Yaskawa INFORM job: A_ROOF_UPPER_0614_2_PAINT_14.JBI

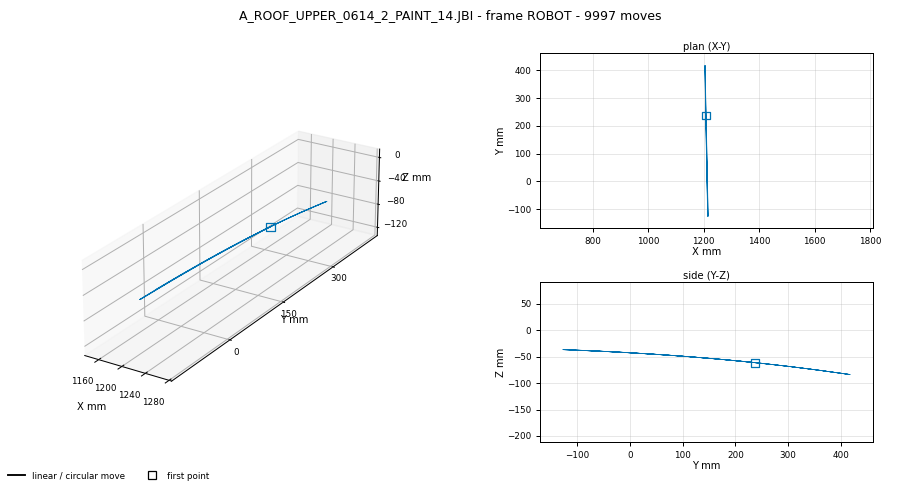
[picture p0: tool path of A_ROOF_UPPER_0614_2_PAINT_14.JBI in frame ROBOT, 9997 of 9997 moves have a stored position in this frame; points joined in program order, loops and branches not executed]
/JOB
//NAME A_ROOF_UPPER_0614_2_PAINT14
//POS
///NPOS 9997,0,0,0,0,0
///TOOL 1
///USER 0
///POSTYPE ROBOT
///RECTAN
///RCONF 1,0,0,0,0,0,0,0,0,0,0,0,0,0,0,0,0,0,0,0,0,0,0,0
C00000=1208.790,237.146,-61.145,-177.184,6.593,148.379
C00001=1208.795,236.875,-61.116,-177.187,6.591,148.380
C00002=1208.800,236.604,-61.089,-177.189,6.589,148.380
C00003=1208.804,236.355,-61.063,-177.193,6.586,148.380
C00004=1208.809,236.106,-61.037,-177.195,6.584,148.380
C00005=1208.814,235.857,-61.011,-177.197,6.582,148.381
C00006=1208.818,235.609,-60.985,-177.200,6.580,148.381
C00007=1208.823,235.360,-60.960,-177.202,6.578,148.381
C00008=1208.827,235.111,-60.934,-177.205,6.576,148.381
C00009=1208.831,234.863,-60.908,-177.207,6.575,148.382
C00010=1208.836,234.614,-60.883,-177.211,6.572,148.382
C00011=1208.840,234.366,-60.857,-177.213,6.570,148.382
C00012=1208.844,234.117,-60.831,-177.215,6.568,148.382
C00013=1208.850,233.868,-60.805,-177.218,6.566,148.383
C00014=1208.854,233.620,-60.780,-177.220,6.564,148.383
C00015=1208.858,233.371,-60.754,-177.223,6.562,148.383
C00016=1208.863,233.123,-60.728,-177.225,6.560,148.384
C00017=1208.867,232.874,-60.703,-177.228,6.558,148.384
C00018=1208.872,232.625,-60.677,-177.231,6.555,148.384
C00019=1208.876,232.377,-60.652,-177.233,6.553,148.384
C00020=1208.881,232.128,-60.626,-177.236,6.552,148.385
C00021=1208.885,231.879,-60.600,-177.239,6.550,148.385
C00022=1208.890,231.631,-60.575,-177.241,6.548,148.385
C00023=1208.894,231.383,-60.549,-177.243,6.546,148.385
C00024=1208.898,231.134,-60.523,-177.246,6.544,148.386
C00025=1208.903,230.885,-60.499,-177.248,6.542,148.386
C00026=1208.908,230.636,-60.473,-177.251,6.539,148.386
C00027=1208.912,230.387,-60.447,-177.254,6.537,148.386
C00028=1208.917,230.139,-60.422,-177.257,6.535,148.387
C00029=1208.921,229.890,-60.396,-177.259,6.533,148.387
C00030=1208.925,229.641,-60.371,-177.261,6.531,148.387
C00031=1208.930,229.393,-60.345,-177.264,6.529,148.387
C00032=1208.934,229.144,-60.320,-177.267,6.528,148.388
C00033=1208.939,228.896,-60.294,-177.269,6.526,148.388
C00034=1208.944,228.647,-60.269,-177.272,6.524,148.388
C00035=1208.948,228.398,-60.244,-177.274,6.522,148.388
C00036=1208.953,228.150,-60.218,-177.277,6.519,148.389
C00037=1208.957,227.901,-60.192,-177.280,6.517,148.389
C00038=1208.962,227.652,-60.168,-177.282,6.515,148.389
C00039=1208.966,227.403,-60.142,-177.285,6.513,148.390
C00040=1208.971,227.155,-60.117,-177.287,6.511,148.390
C00041=1208.975,226.906,-60.092,-177.290,6.510,148.390
C00042=1208.979,226.657,-60.066,-177.292,6.507,148.390
C00043=1208.984,226.409,-60.041,-177.295,6.505,148.391
C00044=1208.989,226.160,-60.016,-177.297,6.504,148.391
C00045=1208.993,225.912,-59.991,-177.300,6.502,148.391
C00046=1208.998,225.663,-59.965,-177.303,6.500,148.392
C00047=1209.003,225.414,-59.940,-177.305,6.497,148.392
C00048=1209.007,225.165,-59.914,-177.308,6.495,148.392
C00049=1209.011,224.917,-59.890,-177.311,6.493,148.392
C00050=1209.016,224.668,-59.865,-177.313,6.491,148.393
C00051=1209.020,224.419,-59.840,-177.316,6.490,148.393
C00052=1209.025,224.171,-59.814,-177.318,6.487,148.393
C00053=1209.029,223.922,-59.788,-177.321,6.486,148.393
C00054=1209.034,223.673,-59.764,-177.323,6.484,148.394
C00055=1209.038,223.425,-59.739,-177.326,6.482,148.394
C00056=1209.043,223.176,-59.714,-177.329,6.480,148.394
C00057=1209.047,222.927,-59.688,-177.331,6.478,148.394
C00058=1209.052,222.678,-59.664,-177.333,6.476,148.395
C00059=1209.056,222.429,-59.639,-177.336,6.474,148.395
C00060=1209.061,222.181,-59.614,-177.339,6.472,148.395
C00061=1209.066,221.932,-59.589,-177.342,6.470,148.396
C00062=1209.070,221.684,-59.563,-177.345,6.468,148.396
C00063=1209.075,221.435,-59.539,-177.347,6.466,148.396
C00064=1209.079,221.186,-59.513,-177.349,6.464,148.397
C00065=1209.084,220.938,-59.489,-177.352,6.462,148.397
C00066=1209.088,220.689,-59.464,-177.355,6.460,148.397
C00067=1209.093,220.440,-59.439,-177.357,6.458,148.398
C00068=1209.097,220.191,-59.414,-177.360,6.456,148.398
C00069=1209.102,219.943,-59.389,-177.362,6.454,148.398
C00070=1209.106,219.694,-59.364,-177.365,6.452,148.398
C00071=1209.111,219.445,-59.339,-177.367,6.451,148.399
C00072=1209.116,219.197,-59.314,-177.370,6.449,148.399
C00073=1209.120,218.948,-59.290,-177.373,6.447,148.399
C00074=1209.125,218.699,-59.265,-177.375,6.445,148.400
C00075=1209.128,218.450,-59.240,-177.377,6.443,148.400
C00076=1209.133,218.202,-59.215,-177.380,6.441,148.400
C00077=1209.138,217.952,-59.190,-177.383,6.438,148.400
C00078=1209.142,217.704,-59.166,-177.386,6.437,148.401
C00079=1209.147,217.455,-59.141,-177.389,6.435,148.401
C00080=1209.152,217.207,-59.116,-177.391,6.433,148.401
C00081=1209.156,216.958,-59.091,-177.394,6.431,148.402
C00082=1209.160,216.709,-59.066,-177.396,6.429,148.402
C00083=1209.165,216.460,-59.042,-177.399,6.427,148.402
C00084=1209.170,216.212,-59.017,-177.401,6.425,148.402
C00085=1209.173,215.963,-58.993,-177.404,6.423,148.403
C00086=1209.179,215.714,-58.968,-177.407,6.422,148.403
C00087=1209.184,215.466,-58.943,-177.409,6.420,148.403
C00088=1209.188,215.217,-58.919,-177.412,6.418,148.404
C00089=1209.193,214.968,-58.894,-177.414,6.416,148.404
C00090=1209.197,214.719,-58.870,-177.417,6.414,148.404
C00091=1209.201,214.471,-58.844,-177.419,6.412,148.405
C00092=1209.206,214.222,-58.820,-177.422,6.410,148.405
C00093=1209.211,213.973,-58.796,-177.425,6.408,148.405
C00094=1209.215,213.724,-58.771,-177.427,6.406,148.406
C00095=1209.220,213.476,-58.746,-177.430,6.405,148.406
C00096=1209.224,213.227,-58.722,-177.432,6.403,148.406
C00097=1209.229,212.978,-58.697,-177.435,6.401,148.407
C00098=1209.233,212.729,-58.673,-177.438,6.399,148.407
C00099=1209.238,212.481,-58.649,-177.440,6.397,148.407
C00100=1209.242,212.232,-58.624,-177.443,6.395,148.407
C00101=1209.247,211.983,-58.599,-177.445,6.393,148.408
C00102=1209.252,211.734,-58.575,-177.448,6.391,148.408
C00103=1209.257,211.464,-58.549,-177.451,6.389,148.408
C00104=1209.261,211.193,-58.522,-177.454,6.387,148.409
C00105=1209.266,210.923,-58.496,-177.456,6.385,148.409
C00106=1209.271,210.653,-58.469,-177.459,6.384,148.410
C00107=1209.276,210.404,-58.445,-177.462,6.381,148.410
C00108=1209.280,210.155,-58.420,-177.464,6.380,148.410
C00109=1209.284,209.906,-58.396,-177.467,6.378,148.410
C00110=1209.290,209.658,-58.372,-177.470,6.376,148.411
C00111=1209.294,209.409,-58.348,-177.472,6.374,148.411
C00112=1209.299,209.159,-58.323,-177.475,6.372,148.411
C00113=1209.303,208.911,-58.299,-177.477,6.370,148.412
C00114=1209.308,208.662,-58.275,-177.480,6.369,148.412
C00115=1209.313,208.414,-58.250,-177.483,6.367,148.412
C00116=1209.316,208.165,-58.226,-177.485,6.365,148.413
C00117=1209.321,207.916,-58.202,-177.488,6.363,148.413
C00118=1209.326,207.667,-58.178,-177.491,6.361,148.413
C00119=1209.331,207.418,-58.154,-177.493,6.359,148.414
C00120=1209.335,207.170,-58.130,-177.495,6.357,148.414
C00121=1209.340,206.921,-58.105,-177.498,6.355,148.414
C00122=1209.344,206.672,-58.081,-177.501,6.354,148.415
C00123=1209.349,206.423,-58.057,-177.503,6.352,148.415
C00124=1209.353,206.175,-58.033,-177.506,6.350,148.415
C00125=1209.358,205.926,-58.009,-177.509,6.348,148.416
C00126=1209.362,205.677,-57.984,-177.511,6.346,148.416
C00127=1209.367,205.428,-57.961,-177.514,6.344,148.416
C00128=1209.371,205.179,-57.937,-177.517,6.343,148.417
C00129=1209.376,204.931,-57.912,-177.519,6.341,148.417
C00130=1209.381,204.682,-57.889,-177.522,6.339,148.417
C00131=1209.385,204.433,-57.865,-177.525,6.337,148.418
C00132=1209.389,204.184,-57.840,-177.527,6.335,148.418
C00133=1209.395,203.935,-57.816,-177.530,6.333,148.418
C00134=1209.399,203.686,-57.792,-177.533,6.332,148.419
C00135=1209.404,203.437,-57.769,-177.535,6.330,148.419
C00136=1209.408,203.189,-57.745,-177.538,6.328,148.419
C00137=1209.412,202.941,-57.721,-177.540,6.326,148.420
C00138=1209.418,202.691,-57.697,-177.543,6.324,148.420
C00139=1209.422,202.443,-57.673,-177.546,6.322,148.420
C00140=1209.426,202.193,-57.649,-177.548,6.320,148.420
C00141=1209.431,201.945,-57.625,-177.551,6.319,148.421
C00142=1209.435,201.696,-57.601,-177.553,6.317,148.421
C00143=1209.440,201.447,-57.577,-177.556,6.315,148.421
C00144=1209.444,201.199,-57.553,-177.558,6.314,148.422
C00145=1209.450,200.949,-57.529,-177.561,6.312,148.422
C00146=1209.454,200.701,-57.505,-177.563,6.310,148.422
C00147=1209.459,200.452,-57.482,-177.566,6.308,148.423
C00148=1209.463,200.204,-57.458,-177.569,6.307,148.423
C00149=1209.468,199.955,-57.434,-177.571,6.305,148.424
C00150=1209.472,199.705,-57.411,-177.574,6.303,148.424
C00151=1209.476,199.456,-57.387,-177.576,6.301,148.424
C00152=1209.481,199.207,-57.363,-177.579,6.299,148.425
C00153=1209.486,198.959,-57.339,-177.582,6.297,148.425
C00154=1209.490,198.710,-57.316,-177.584,6.296,148.425
C00155=1209.495,198.462,-57.292,-177.587,6.294,148.426
C00156=1209.499,198.213,-57.268,-177.590,6.292,148.426
C00157=1209.504,197.963,-57.245,-177.592,6.290,148.426
C00158=1209.508,197.715,-57.221,-177.595,6.288,148.427
C00159=1209.513,197.466,-57.198,-177.597,6.287,148.427
C00160=1209.518,197.217,-57.174,-177.600,6.285,148.427
C00161=1209.523,196.968,-57.150,-177.602,6.284,148.428
C00162=1209.528,196.719,-57.126,-177.605,6.282,148.428
C00163=1209.532,196.471,-57.104,-177.608,6.280,148.428
C00164=1209.536,196.222,-57.079,-177.610,6.278,148.429
C00165=1209.541,195.973,-57.056,-177.613,6.276,148.429
C00166=1209.545,195.724,-57.033,-177.616,6.274,148.429
C00167=1209.550,195.476,-57.009,-177.618,6.273,148.430
C00168=1209.554,195.227,-56.985,-177.621,6.271,148.430
C00169=1209.559,194.978,-56.962,-177.624,6.269,148.430
C00170=1209.564,194.729,-56.939,-177.626,6.268,148.431
C00171=1209.568,194.480,-56.914,-177.628,6.266,148.431
C00172=1209.573,194.231,-56.891,-177.631,6.264,148.432
C00173=1209.578,193.982,-56.868,-177.634,6.263,148.432
C00174=1209.582,193.733,-56.844,-177.636,6.261,148.432
C00175=1209.587,193.484,-56.821,-177.639,6.259,148.433
C00176=1209.591,193.236,-56.797,-177.642,6.257,148.433
C00177=1209.596,192.987,-56.774,-177.644,6.255,148.433
C00178=1209.601,192.738,-56.750,-177.647,6.253,148.434
C00179=1209.605,192.489,-56.728,-177.649,6.252,148.434
C00180=1209.610,192.240,-56.704,-177.652,6.251,148.435
C00181=1209.615,191.991,-56.681,-177.655,6.249,148.435
C00182=1209.620,191.742,-56.658,-177.657,6.247,148.435
C00183=1209.624,191.493,-56.634,-177.660,6.245,148.436
C00184=1209.629,191.245,-56.610,-177.663,6.244,148.436
C00185=1209.633,190.996,-56.587,-177.665,6.242,148.436
C00186=1209.637,190.747,-56.564,-177.668,6.240,148.437
C00187=1209.642,190.498,-56.541,-177.670,6.239,148.437
C00188=1209.647,190.249,-56.518,-177.673,6.237,148.437
C00189=1209.651,190.000,-56.494,-177.675,6.235,148.438
C00190=1209.656,189.751,-56.471,-177.678,6.233,148.438
C00191=1209.661,189.503,-56.448,-177.681,6.232,148.438
C00192=1209.665,189.254,-56.425,-177.683,6.230,148.439
C00193=1209.670,189.005,-56.402,-177.686,6.228,148.439
C00194=1209.675,188.756,-56.378,-177.689,6.226,148.439
C00195=1209.679,188.507,-56.355,-177.691,6.225,148.440
C00196=1209.683,188.258,-56.332,-177.693,6.223,148.440
C00197=1209.688,188.009,-56.309,-177.696,6.222,148.441
C00198=1209.693,187.760,-56.285,-177.699,6.220,148.441
C00199=1209.698,187.512,-56.262,-177.701,6.218,148.441
C00200=1209.702,187.262,-56.240,-177.704,6.216,148.442
C00201=1209.707,187.013,-56.217,-177.707,6.215,148.442
C00202=1209.712,186.764,-56.194,-177.709,6.214,148.443
C00203=1209.716,186.516,-56.171,-177.712,6.212,148.443
C00204=1209.720,186.267,-56.148,-177.715,6.210,148.443
C00205=1209.726,186.018,-56.125,-177.717,6.208,148.444
C00206=1209.730,185.770,-56.102,-177.720,6.206,148.444
C00207=1209.735,185.500,-56.077,-177.723,6.205,148.444
C00208=1209.740,185.230,-56.052,-177.725,6.203,148.445
C00209=1209.745,184.961,-56.027,-177.728,6.201,148.445
C00210=1209.750,184.691,-56.002,-177.731,6.199,148.446
C00211=1209.755,184.442,-55.979,-177.734,6.198,148.446
C00212=1209.759,184.193,-55.956,-177.736,6.196,148.446
C00213=1209.764,183.943,-55.934,-177.738,6.195,148.447
C00214=1209.768,183.695,-55.911,-177.741,6.193,148.447
C00215=1209.773,183.446,-55.888,-177.744,6.191,148.447
C00216=1209.778,183.197,-55.864,-177.746,6.189,148.448
C00217=1209.782,182.948,-55.842,-177.750,6.188,148.448
C00218=1209.787,182.699,-55.819,-177.752,6.186,148.449
C00219=1209.791,182.451,-55.797,-177.754,6.185,148.449
C00220=1209.796,182.202,-55.773,-177.757,6.183,148.449
C00221=1209.801,181.952,-55.751,-177.760,6.181,148.450
C00222=1209.805,181.704,-55.728,-177.762,6.180,148.450
C00223=1209.810,181.455,-55.705,-177.765,6.178,148.450
C00224=1209.815,181.206,-55.683,-177.767,6.177,148.451
C00225=1209.819,180.957,-55.659,-177.770,6.175,148.451
C00226=1209.823,180.708,-55.637,-177.772,6.173,148.452
C00227=1209.829,180.459,-55.614,-177.775,6.172,148.452
C00228=1209.833,180.210,-55.592,-177.778,6.170,148.453
C00229=1209.838,179.961,-55.569,-177.781,6.168,148.453
C00230=1209.842,179.713,-55.547,-177.783,6.167,148.453
C00231=1209.847,179.464,-55.523,-177.786,6.165,148.454
C00232=1209.851,179.214,-55.501,-177.788,6.163,148.454
C00233=1209.856,178.965,-55.478,-177.791,6.162,148.454
C00234=1209.861,178.717,-55.456,-177.793,6.161,148.455
C00235=1209.866,178.468,-55.433,-177.796,6.159,148.455
C00236=1209.870,178.218,-55.411,-177.799,6.157,148.456
C00237=1209.875,177.970,-55.388,-177.801,6.155,148.456
C00238=1209.880,177.721,-55.366,-177.804,6.154,148.456
C00239=1209.884,177.472,-55.342,-177.806,6.153,148.457
C00240=1209.889,177.223,-55.321,-177.809,6.151,148.457
C00241=1209.894,176.974,-55.297,-177.811,6.149,148.457
C00242=1209.898,176.725,-55.275,-177.814,6.147,148.458
C00243=1209.903,176.477,-55.253,-177.817,6.146,148.458
C00244=1209.908,176.227,-55.230,-177.819,6.145,148.459
C00245=1209.912,175.978,-55.207,-177.822,6.143,148.459
C00246=1209.917,175.729,-55.185,-177.825,6.141,148.460
C00247=1209.921,175.481,-55.162,-177.827,6.139,148.460
C00248=1209.926,175.232,-55.141,-177.829,6.138,148.460
C00249=1209.931,174.982,-55.118,-177.832,6.137,148.461
C00250=1209.935,174.734,-55.095,-177.835,6.135,148.461
C00251=1209.940,174.485,-55.074,-177.838,6.133,148.462
C00252=1209.945,174.235,-55.051,-177.840,6.132,148.462
C00253=1209.949,173.987,-55.028,-177.843,6.130,148.462
C00254=1209.954,173.738,-55.006,-177.845,6.129,148.463
C00255=1209.959,173.488,-54.984,-177.848,6.127,148.463
C00256=1209.963,173.240,-54.962,-177.851,6.125,148.463
C00257=1209.968,172.991,-54.939,-177.853,6.124,148.464
C00258=1209.973,172.742,-54.917,-177.856,6.123,148.464
C00259=1209.977,172.493,-54.894,-177.859,6.121,148.465
C00260=1209.981,172.244,-54.872,-177.861,6.119,148.465
C00261=1209.987,171.995,-54.850,-177.863,6.118,148.465
C00262=1209.991,171.746,-54.827,-177.866,6.116,148.466
C00263=1209.996,171.498,-54.806,-177.869,6.115,148.466
C00264=1210.001,171.248,-54.783,-177.872,6.113,148.467
C00265=1210.006,170.999,-54.761,-177.874,6.112,148.467
C00266=1210.010,170.750,-54.739,-177.877,6.110,148.468
C00267=1210.014,170.501,-54.717,-177.879,6.108,148.468
C00268=1210.020,170.252,-54.694,-177.881,6.107,148.468
C00269=1210.024,170.003,-54.672,-177.884,6.106,148.469
C00270=1210.029,169.754,-54.650,-177.887,6.104,148.469
C00271=1210.033,169.505,-54.628,-177.890,6.102,148.470
C00272=1210.037,169.257,-54.606,-177.892,6.101,148.470
C00273=1210.042,169.007,-54.583,-177.895,6.099,148.470
C00274=1210.047,168.759,-54.562,-177.897,6.098,148.471
C00275=1210.052,168.509,-54.540,-177.900,6.096,148.471
C00276=1210.056,168.261,-54.518,-177.902,6.095,148.472
C00277=1210.061,168.011,-54.496,-177.905,6.093,148.472
C00278=1210.066,167.762,-54.474,-177.908,6.091,148.472
C00279=1210.071,167.513,-54.452,-177.910,6.090,148.473
C00280=1210.076,167.264,-54.430,-177.913,6.089,148.473
C00281=1210.080,167.015,-54.408,-177.916,6.087,148.474
C00282=1210.084,166.767,-54.385,-177.918,6.085,148.474
C00283=1210.089,166.518,-54.363,-177.920,6.084,148.475
C00284=1210.094,166.269,-54.341,-177.923,6.083,148.475
C00285=1210.098,166.019,-54.319,-177.926,6.081,148.475
C00286=1210.103,165.771,-54.297,-177.929,6.079,148.476
C00287=1210.108,165.521,-54.275,-177.931,6.078,148.476
C00288=1210.112,165.273,-54.254,-177.934,6.077,148.477
C00289=1210.117,165.024,-54.232,-177.936,6.075,148.477
C00290=1210.122,164.775,-54.210,-177.939,6.074,148.478
C00291=1210.126,164.526,-54.188,-177.942,6.072,148.478
C00292=1210.131,164.276,-54.167,-177.944,6.070,148.478
C00293=1210.136,164.028,-54.145,-177.946,6.070,148.479
C00294=1210.140,163.778,-54.123,-177.950,6.068,148.479
C00295=1210.145,163.530,-54.102,-177.952,6.066,148.480
C00296=1210.150,163.281,-54.080,-177.954,6.065,148.480
C00297=1210.154,163.032,-54.058,-177.957,6.063,148.480
C00298=1210.160,162.783,-54.036,-177.960,6.062,148.481
C00299=1210.164,162.533,-54.013,-177.963,6.060,148.481
C00300=1210.169,162.285,-53.992,-177.965,6.059,148.482
C00301=1210.173,162.035,-53.970,-177.968,6.057,148.482
C00302=1210.178,161.786,-53.949,-177.970,6.056,148.482
C00303=1210.183,161.537,-53.927,-177.973,6.055,148.483
C00304=1210.188,161.288,-53.905,-177.976,6.053,148.483
C00305=1210.192,161.039,-53.883,-177.978,6.051,148.484
C00306=1210.197,160.791,-53.862,-177.980,6.050,148.484
C00307=1210.201,160.542,-53.840,-177.983,6.049,148.485
C00308=1210.206,160.293,-53.819,-177.986,6.047,148.485
C00309=1210.210,160.043,-53.797,-177.988,6.046,148.486
C00310=1210.215,159.795,-53.776,-177.991,6.044,148.486
C00311=1210.221,159.525,-53.752,-177.994,6.043,148.487
C00312=1210.225,159.256,-53.729,-177.997,6.041,148.487
C00313=1210.231,158.987,-53.705,-177.999,6.039,148.487
C00314=1210.236,158.718,-53.682,-178.003,6.038,148.488
C00315=1210.240,158.470,-53.661,-178.005,6.037,148.488
C00316=1210.245,158.220,-53.640,-178.007,6.035,148.489
C00317=1210.250,157.971,-53.618,-178.010,6.034,148.489
C00318=1210.254,157.722,-53.596,-178.013,6.033,148.490
C00319=1210.259,157.474,-53.575,-178.015,6.031,148.490
C00320=1210.264,157.224,-53.553,-178.017,6.030,148.490
C00321=1210.269,156.975,-53.532,-178.020,6.028,148.491
C00322=1210.274,156.726,-53.511,-178.023,6.027,148.491
C00323=1210.278,156.477,-53.488,-178.025,6.026,148.492
C00324=1210.282,156.228,-53.467,-178.028,6.024,148.492
C00325=1210.288,155.979,-53.446,-178.031,6.022,148.493
C00326=1210.292,155.730,-53.424,-178.033,6.021,148.493
C00327=1210.297,155.481,-53.403,-178.036,6.020,148.493
C00328=1210.302,155.232,-53.382,-178.039,6.018,148.494
C00329=1210.307,154.983,-53.360,-178.041,6.017,148.494
C00330=1210.311,154.733,-53.339,-178.044,6.015,148.495
C00331=1210.315,154.485,-53.318,-178.046,6.013,148.495
C00332=1210.321,154.236,-53.297,-178.049,6.013,148.496
C00333=1210.325,153.987,-53.275,-178.052,6.011,148.496
C00334=1210.330,153.737,-53.254,-178.054,6.010,148.497
C00335=1210.334,153.489,-53.233,-178.057,6.008,148.497
C00336=1210.339,153.239,-53.212,-178.060,6.007,148.498
C00337=1210.344,152.991,-53.190,-178.062,6.006,148.498
C00338=1210.349,152.741,-53.169,-178.064,6.004,148.498
C00339=1210.353,152.492,-53.148,-178.068,6.003,148.499
C00340=1210.358,152.243,-53.127,-178.070,6.002,148.499
C00341=1210.363,151.995,-53.105,-178.072,6.000,148.500
C00342=1210.368,151.745,-53.084,-178.074,5.999,148.500
C00343=1210.372,151.496,-53.062,-178.078,5.997,148.501
C00344=1210.377,151.247,-53.041,-178.080,5.996,148.501
C00345=1210.382,150.998,-53.020,-178.082,5.995,148.502
C00346=1210.386,150.749,-52.999,-178.086,5.993,148.502
C00347=1210.391,150.499,-52.978,-178.088,5.991,148.502
C00348=1210.396,150.251,-52.956,-178.090,5.990,148.503
C00349=1210.400,150.002,-52.936,-178.093,5.989,148.503
C00350=1210.405,149.753,-52.915,-178.096,5.988,148.504
C00351=1210.410,149.504,-52.893,-178.098,5.986,148.504
C00352=1210.414,149.255,-52.873,-178.101,5.984,148.505
C00353=1210.419,149.005,-52.852,-178.104,5.984,148.505
C00354=1210.424,148.756,-52.830,-178.106,5.982,148.506
C00355=1210.428,148.507,-52.810,-178.108,5.981,148.506
C00356=1210.434,148.258,-52.789,-178.112,5.980,148.507
C00357=1210.439,148.009,-52.768,-178.114,5.978,148.507
C00358=1210.443,147.761,-52.747,-178.116,5.977,148.507
C00359=1210.447,147.511,-52.725,-178.119,5.975,148.508
C00360=1210.452,147.262,-52.705,-178.122,5.974,148.508
C00361=1210.457,147.013,-52.683,-178.124,5.973,148.509
C00362=1210.462,146.764,-52.662,-178.127,5.972,148.509
C00363=1210.466,146.515,-52.642,-178.130,5.970,148.510
C00364=1210.472,146.266,-52.621,-178.132,5.968,148.510
C00365=1210.476,146.017,-52.601,-178.135,5.968,148.511
C00366=1210.481,145.768,-52.579,-178.137,5.966,148.511
C00367=1210.485,145.518,-52.558,-178.140,5.965,148.512
C00368=1210.490,145.269,-52.537,-178.143,5.963,148.512
C00369=1210.495,145.020,-52.516,-178.145,5.962,148.513
C00370=1210.499,144.771,-52.496,-178.148,5.961,148.513
C00371=1210.505,144.522,-52.475,-178.150,5.959,148.513
C00372=1210.509,144.273,-52.454,-178.153,5.958,148.514
C00373=1210.514,144.024,-52.433,-178.155,5.957,148.514
C00374=1210.518,143.775,-52.412,-178.158,5.956,148.515
C00375=1210.524,143.526,-52.391,-178.161,5.954,148.515
C00376=1210.528,143.277,-52.371,-178.163,5.952,148.516
C00377=1210.533,143.028,-52.350,-178.166,5.952,148.516
C00378=1210.537,142.778,-52.329,-178.169,5.950,148.517
C00379=1210.542,142.529,-52.308,-178.171,5.949,148.517
C00380=1210.547,142.280,-52.288,-178.174,5.947,148.518
C00381=1210.552,142.031,-52.267,-178.176,5.946,148.518
C00382=1210.556,141.782,-52.247,-178.179,5.945,148.519
C00383=1210.561,141.533,-52.226,-178.181,5.944,148.519
C00384=1210.566,141.283,-52.205,-178.184,5.942,148.520
C00385=1210.570,141.034,-52.185,-178.187,5.940,148.520
C00386=1210.575,140.785,-52.164,-178.189,5.940,148.521
C00387=1210.580,140.536,-52.144,-178.192,5.938,148.521
C00388=1210.585,140.287,-52.123,-178.194,5.937,148.521
C00389=1210.589,140.038,-52.102,-178.197,5.936,148.522
C00390=1210.594,139.789,-52.082,-178.199,5.935,148.522
C00391=1210.599,139.540,-52.061,-178.202,5.933,148.523
C00392=1210.604,139.291,-52.041,-178.205,5.932,148.523
C00393=1210.608,139.042,-52.020,-178.207,5.930,148.524
C00394=1210.613,138.793,-51.999,-178.210,5.930,148.524
C00395=1210.618,138.544,-51.979,-178.213,5.928,148.525
C00396=1210.623,138.294,-51.958,-178.215,5.927,148.525
C00397=1210.627,138.045,-51.938,-178.218,5.926,148.526
C00398=1210.632,137.797,-51.917,-178.221,5.924,148.526
C00399=1210.637,137.547,-51.896,-178.223,5.923,148.527
C00400=1210.642,137.298,-51.877,-178.226,5.921,148.527
C00401=1210.646,137.049,-51.856,-178.228,5.921,148.528
C00402=1210.651,136.799,-51.835,-178.231,5.919,148.528
C00403=1210.656,136.551,-51.815,-178.233,5.918,148.529
C00404=1210.660,136.302,-51.794,-178.236,5.916,148.529
C00405=1210.665,136.052,-51.773,-178.239,5.916,148.530
C00406=1210.670,135.803,-51.754,-178.241,5.914,148.530
C00407=1210.675,135.555,-51.734,-178.244,5.913,148.531
C00408=1210.679,135.306,-51.713,-178.246,5.912,148.531
C00409=1210.685,135.056,-51.692,-178.249,5.911,148.531
C00410=1210.689,134.807,-51.673,-178.252,5.909,148.532
C00411=1210.694,134.558,-51.652,-178.254,5.908,148.532
C00412=1210.698,134.309,-51.632,-178.257,5.906,148.533
C00413=1210.703,134.060,-51.611,-178.259,5.906,148.533
C00414=1210.708,133.810,-51.591,-178.262,5.904,148.534
C00415=1210.713,133.542,-51.569,-178.265,5.903,148.534
C00416=1210.718,133.273,-51.548,-178.267,5.902,148.535
C00417=1210.724,133.005,-51.526,-178.270,5.900,148.535
C00418=1210.729,132.736,-51.505,-178.273,5.899,148.536
C00419=1210.734,132.487,-51.484,-178.276,5.898,148.536
C00420=1210.738,132.238,-51.463,-178.278,5.896,148.537
C00421=1210.743,131.988,-51.444,-178.281,5.895,148.537
C00422=1210.747,131.739,-51.423,-178.284,5.894,148.538
C00423=1210.752,131.490,-51.403,-178.286,5.893,148.538
C00424=1210.757,131.241,-51.383,-178.289,5.891,148.539
C00425=1210.762,130.992,-51.362,-178.291,5.890,148.539
C00426=1210.767,130.743,-51.343,-178.294,5.889,148.540
C00427=1210.772,130.494,-51.322,-178.296,5.888,148.540
C00428=1210.776,130.245,-51.302,-178.299,5.886,148.541
C00429=1210.781,129.995,-51.282,-178.302,5.885,148.541
C00430=1210.785,129.746,-51.262,-178.304,5.885,148.542
C00431=1210.790,129.497,-51.242,-178.307,5.883,148.542
C00432=1210.796,129.248,-51.222,-178.309,5.882,148.543
C00433=1210.800,128.999,-51.202,-178.312,5.881,148.543
C00434=1210.805,128.750,-51.182,-178.314,5.880,148.544
C00435=1210.810,128.500,-51.162,-178.317,5.878,148.544
C00436=1210.814,128.251,-51.142,-178.320,5.877,148.545
C00437=1210.819,128.001,-51.122,-178.323,5.876,148.545
C00438=1210.824,127.753,-51.102,-178.325,5.875,148.546
C00439=1210.829,127.504,-51.082,-178.327,5.873,148.546
C00440=1210.833,127.255,-51.062,-178.330,5.872,148.547
C00441=1210.838,127.005,-51.042,-178.333,5.871,148.547
C00442=1210.842,126.756,-51.022,-178.335,5.870,148.548
C00443=1210.848,126.507,-51.003,-178.338,5.868,148.548
C00444=1210.852,126.258,-50.982,-178.341,5.868,148.549
C00445=1210.857,126.009,-50.963,-178.343,5.866,148.549
C00446=1210.861,125.759,-50.943,-178.345,5.865,148.550
C00447=1210.867,125.511,-50.923,-178.348,5.864,148.550
C00448=1210.871,125.261,-50.903,-178.351,5.863,148.551
C00449=1210.876,125.013,-50.883,-178.353,5.862,148.551
C00450=1210.880,124.763,-50.863,-178.356,5.860,148.552
C00451=1210.886,124.514,-50.844,-178.359,5.860,148.552
C00452=1210.890,124.265,-50.824,-178.361,5.858,148.553
C00453=1210.895,124.016,-50.804,-178.364,5.857,148.553
C00454=1210.900,123.766,-50.784,-178.367,5.855,148.554
C00455=1210.905,123.518,-50.764,-178.369,5.855,148.554
C00456=1210.909,123.268,-50.745,-178.371,5.854,148.555
C00457=1210.914,123.019,-50.725,-178.374,5.852,148.555
C00458=1210.919,122.769,-50.705,-178.377,5.851,148.556
C00459=1210.924,122.521,-50.685,-178.379,5.850,148.556
C00460=1210.929,122.271,-50.666,-178.382,5.849,148.557
C00461=1210.934,122.022,-50.646,-178.385,5.847,148.557
C00462=1210.939,121.773,-50.626,-178.387,5.847,148.558
C00463=1210.943,121.524,-50.606,-178.389,5.846,148.558
C00464=1210.948,121.274,-50.587,-178.393,5.844,148.559
C00465=1210.953,121.025,-50.567,-178.395,5.843,148.559
C00466=1210.957,120.776,-50.548,-178.398,5.842,148.560
C00467=1210.962,120.527,-50.528,-178.400,5.841,148.560
C00468=1210.967,120.278,-50.508,-178.403,5.839,148.561
C00469=1210.972,120.029,-50.489,-178.405,5.838,148.561
C00470=1210.977,119.779,-50.469,-178.408,5.838,148.562
C00471=1210.981,119.530,-50.450,-178.411,5.836,148.562
C00472=1210.986,119.281,-50.430,-178.413,5.835,148.563
C00473=1210.991,119.032,-50.410,-178.416,5.834,148.563
C00474=1210.995,118.783,-50.391,-178.418,5.833,148.564
C00475=1211.001,118.534,-50.372,-178.421,5.831,148.564
C00476=1211.005,118.284,-50.352,-178.423,5.830,148.565
C00477=1211.010,118.035,-50.332,-178.426,5.830,148.566
C00478=1211.015,117.786,-50.313,-178.429,5.828,148.566
C00479=1211.020,117.536,-50.294,-178.431,5.827,148.567
C00480=1211.025,117.288,-50.275,-178.434,5.826,148.567
C00481=1211.029,117.039,-50.254,-178.436,5.825,148.568
C00482=1211.034,116.789,-50.235,-178.439,5.824,148.568
C00483=1211.039,116.540,-50.216,-178.442,5.823,148.569
C00484=1211.043,116.291,-50.196,-178.444,5.822,148.569
C00485=1211.049,116.042,-50.177,-178.447,5.820,148.570
C00486=1211.053,115.792,-50.158,-178.449,5.819,148.570
C00487=1211.058,115.543,-50.138,-178.452,5.819,148.571
C00488=1211.063,115.294,-50.119,-178.455,5.817,148.571
C00489=1211.067,115.045,-50.100,-178.457,5.816,148.572
C00490=1211.073,114.796,-50.080,-178.460,5.815,148.572
C00491=1211.077,114.546,-50.061,-178.462,5.814,148.573
C00492=1211.081,114.297,-50.042,-178.465,5.813,148.573
C00493=1211.087,114.048,-50.022,-178.468,5.812,148.574
C00494=1211.092,113.799,-50.003,-178.470,5.811,148.574
C00495=1211.097,113.550,-49.983,-178.472,5.810,148.575
C00496=1211.101,113.300,-49.965,-178.475,5.808,148.575
C00497=1211.107,113.051,-49.946,-178.478,5.808,148.576
C00498=1211.111,112.801,-49.926,-178.480,5.806,148.576
C00499=1211.115,112.552,-49.907,-178.483,5.805,148.577
C00500=1211.121,112.303,-49.888,-178.485,5.804,148.577
C00501=1211.125,112.054,-49.868,-178.488,5.803,148.578
C00502=1211.130,111.805,-49.849,-178.491,5.802,148.578
C00503=1211.135,111.556,-49.830,-178.493,5.801,148.579
C00504=1211.140,111.307,-49.810,-178.496,5.800,148.580
C00505=1211.144,111.057,-49.792,-178.498,5.799,148.580
C00506=1211.150,110.808,-49.773,-178.502,5.798,148.581
C00507=1211.154,110.559,-49.754,-178.504,5.797,148.581
C00508=1211.159,110.310,-49.734,-178.506,5.796,148.582
C00509=1211.164,110.060,-49.715,-178.509,5.794,148.582
C00510=1211.169,109.811,-49.697,-178.512,5.794,148.583
C00511=1211.174,109.562,-49.677,-178.514,5.793,148.583
C00512=1211.179,109.313,-49.658,-178.517,5.791,148.584
C00513=1211.183,109.063,-49.639,-178.519,5.790,148.584
C00514=1211.188,108.815,-49.619,-178.522,5.790,148.585
C00515=1211.193,108.565,-49.601,-178.524,5.788,148.585
C00516=1211.198,108.316,-49.582,-178.527,5.787,148.586
C00517=1211.202,108.067,-49.563,-178.529,5.786,148.586
C00518=1211.208,107.817,-49.544,-178.532,5.785,148.587
C00519=1211.212,107.548,-49.523,-178.535,5.784,148.588
C00520=1211.217,107.281,-49.503,-178.538,5.783,148.588
C00521=1211.222,107.012,-49.483,-178.540,5.782,148.589
C00522=1211.228,106.744,-49.462,-178.543,5.781,148.589
C00523=1211.233,106.494,-49.444,-178.546,5.780,148.590
C00524=1211.238,106.245,-49.424,-178.549,5.778,148.590
C00525=1211.242,105.996,-49.405,-178.551,5.778,148.591
C00526=1211.247,105.746,-49.387,-178.553,5.777,148.591
C00527=1211.252,105.498,-49.368,-178.557,5.775,148.592
C00528=1211.257,105.248,-49.348,-178.559,5.774,148.593
C00529=1211.262,104.999,-49.330,-178.561,5.774,148.593
C00530=1211.267,104.750,-49.311,-178.564,5.772,148.594
C00531=1211.271,104.501,-49.292,-178.567,5.771,148.594
C00532=1211.277,104.251,-49.273,-178.569,5.770,148.595
C00533=1211.281,104.002,-49.254,-178.572,5.769,148.595
C00534=1211.286,103.752,-49.236,-178.575,5.768,148.596
C00535=1211.291,103.504,-49.217,-178.577,5.768,148.596
C00536=1211.296,103.254,-49.198,-178.580,5.766,148.597
C00537=1211.300,103.005,-49.179,-178.582,5.765,148.597
C00538=1211.305,102.755,-49.161,-178.585,5.765,148.598
C00539=1211.310,102.506,-49.142,-178.587,5.763,148.598
C00540=1211.315,102.257,-49.124,-178.590,5.762,148.599
C00541=1211.320,102.008,-49.104,-178.593,5.762,148.600
C00542=1211.325,101.759,-49.086,-178.595,5.761,148.600
C00543=1211.329,101.510,-49.067,-178.598,5.759,148.601
C00544=1211.334,101.260,-49.048,-178.600,5.758,148.601
C00545=1211.339,101.011,-49.030,-178.603,5.758,148.602
C00546=1211.344,100.761,-49.011,-178.605,5.756,148.602
C00547=1211.349,100.512,-48.992,-178.608,5.755,148.603
C00548=1211.353,100.263,-48.974,-178.611,5.755,148.604
C00549=1211.358,100.014,-48.954,-178.613,5.753,148.604
C00550=1211.363,99.765,-48.936,-178.616,5.752,148.605
C00551=1211.368,99.515,-48.919,-178.618,5.752,148.605
C00552=1211.373,99.266,-48.899,-178.621,5.750,148.606
C00553=1211.378,99.017,-48.881,-178.623,5.749,148.606
C00554=1211.382,98.768,-48.862,-178.626,5.749,148.607
C00555=1211.387,98.518,-48.843,-178.629,5.748,148.607
C00556=1211.392,98.269,-48.825,-178.631,5.746,148.608
C00557=1211.397,98.020,-48.807,-178.634,5.746,148.608
C00558=1211.401,97.770,-48.788,-178.636,5.745,148.609
C00559=1211.407,97.521,-48.770,-178.639,5.743,148.609
C00560=1211.411,97.272,-48.751,-178.642,5.743,148.610
C00561=1211.416,97.023,-48.733,-178.644,5.742,148.611
C00562=1211.421,96.773,-48.714,-178.647,5.741,148.611
C00563=1211.426,96.524,-48.695,-178.649,5.739,148.612
C00564=1211.431,96.275,-48.677,-178.652,5.739,148.612
C00565=1211.435,96.025,-48.659,-178.655,5.738,148.613
C00566=1211.441,95.776,-48.640,-178.657,5.736,148.613
C00567=1211.445,95.527,-48.622,-178.660,5.736,148.614
C00568=1211.450,95.278,-48.604,-178.662,5.735,148.614
C00569=1211.455,95.028,-48.585,-178.665,5.734,148.615
C00570=1211.459,94.780,-48.567,-178.668,5.733,148.616
C00571=1211.465,94.530,-48.548,-178.670,5.732,148.616
C00572=1211.470,94.281,-48.530,-178.673,5.731,148.617
C00573=1211.474,94.031,-48.512,-178.675,5.730,148.617
C00574=1211.479,93.782,-48.494,-178.678,5.729,148.618
C00575=1211.484,93.533,-48.475,-178.680,5.728,148.618
C00576=1211.489,93.284,-48.457,-178.683,5.728,148.619
C00577=1211.494,93.034,-48.438,-178.686,5.726,148.619
C00578=1211.499,92.785,-48.420,-178.688,5.725,148.620
C00579=1211.503,92.536,-48.402,-178.691,5.725,148.621
C00580=1211.508,92.286,-48.384,-178.693,5.724,148.621
C00581=1211.513,92.038,-48.366,-178.696,5.722,148.622
C00582=1211.518,91.788,-48.347,-178.699,5.722,148.622
C00583=1211.523,91.539,-48.329,-178.701,5.721,148.623
C00584=1211.528,91.289,-48.311,-178.703,5.720,148.623
C00585=1211.533,91.040,-48.293,-178.706,5.719,148.624
C00586=1211.538,90.791,-48.275,-178.709,5.718,148.624
C00587=1211.542,90.541,-48.256,-178.711,5.717,148.625
C00588=1211.547,90.292,-48.238,-178.714,5.717,148.626
C00589=1211.552,90.043,-48.220,-178.717,5.715,148.626
C00590=1211.557,89.794,-48.202,-178.719,5.714,148.627
C00591=1211.562,89.544,-48.184,-178.722,5.714,148.627
C00592=1211.567,89.295,-48.166,-178.724,5.713,148.628
C00593=1211.572,89.045,-48.148,-178.727,5.711,148.628
C00594=1211.577,88.796,-48.130,-178.729,5.710,148.629
C00595=1211.581,88.547,-48.112,-178.732,5.710,148.630
C00596=1211.586,88.298,-48.094,-178.734,5.709,148.630
C00597=1211.591,88.048,-48.076,-178.737,5.708,148.631
C00598=1211.596,87.799,-48.058,-178.740,5.707,148.631
C00599=1211.601,87.549,-48.039,-178.742,5.706,148.632
C00600=1211.605,87.300,-48.021,-178.745,5.705,148.632
C00601=1211.610,87.051,-48.003,-178.747,5.705,148.633
C00602=1211.615,86.802,-47.985,-178.750,5.703,148.634
C00603=1211.620,86.553,-47.967,-178.753,5.703,148.634
C00604=1211.625,86.303,-47.949,-178.755,5.702,148.635
C00605=1211.630,86.054,-47.931,-178.757,5.701,148.635
C00606=1211.635,85.805,-47.913,-178.760,5.700,148.636
C00607=1211.640,85.556,-47.895,-178.763,5.699,148.636
C00608=1211.644,85.306,-47.877,-178.765,5.698,148.637
C00609=1211.649,85.057,-47.859,-178.768,5.698,148.638
C00610=1211.654,84.807,-47.842,-178.770,5.697,148.638
C00611=1211.659,84.558,-47.824,-178.773,5.695,148.639
C00612=1211.664,84.309,-47.806,-178.776,5.695,148.639
C00613=1211.669,84.060,-47.788,-178.778,5.694,148.640
C00614=1211.674,83.810,-47.770,-178.781,5.693,148.640
C00615=1211.679,83.561,-47.752,-178.783,5.693,148.641
C00616=1211.684,83.311,-47.735,-178.786,5.691,148.642
C00617=1211.689,83.062,-47.717,-178.789,5.690,148.642
C00618=1211.693,82.813,-47.699,-178.791,5.690,148.643
C00619=1211.698,82.564,-47.681,-178.794,5.689,148.643
C00620=1211.702,82.314,-47.663,-178.796,5.687,148.644
C00621=1211.708,82.064,-47.646,-178.799,5.687,148.644
C00622=1211.712,81.815,-47.628,-178.802,5.686,148.645
C00623=1211.718,81.548,-47.609,-178.804,5.686,148.646
C00624=1211.724,81.279,-47.590,-178.807,5.684,148.646
C00625=1211.729,81.011,-47.571,-178.810,5.683,148.647
C00626=1211.734,80.742,-47.551,-178.812,5.683,148.647
C00627=1211.739,80.493,-47.534,-178.815,5.681,148.648
C00628=1211.744,80.243,-47.516,-178.818,5.680,148.649
C00629=1211.748,79.995,-47.499,-178.820,5.680,148.649
C00630=1211.753,79.745,-47.481,-178.823,5.679,148.650
C00631=1211.758,79.496,-47.463,-178.825,5.678,148.650
C00632=1211.763,79.246,-47.445,-178.828,5.677,148.651
C00633=1211.768,78.997,-47.427,-178.831,5.676,148.652
C00634=1211.773,78.747,-47.410,-178.833,5.676,148.652
C00635=1211.777,78.499,-47.393,-178.836,5.675,148.653
C00636=1211.783,78.249,-47.375,-178.838,5.674,148.653
C00637=1211.787,78.000,-47.357,-178.841,5.674,148.654
C00638=1211.792,77.750,-47.340,-178.844,5.672,148.654
C00639=1211.798,77.501,-47.322,-178.846,5.671,148.655
C00640=1211.802,77.252,-47.305,-178.849,5.671,148.656
C00641=1211.807,77.002,-47.288,-178.851,5.670,148.656
C00642=1211.812,76.753,-47.270,-178.854,5.669,148.657
C00643=1211.817,76.504,-47.252,-178.856,5.669,148.657
C00644=1211.821,76.254,-47.235,-178.859,5.667,148.658
C00645=1211.826,76.005,-47.217,-178.862,5.666,148.659
C00646=1211.831,75.755,-47.200,-178.864,5.666,148.659
C00647=1211.836,75.506,-47.182,-178.866,5.665,148.660
C00648=1211.841,75.257,-47.165,-178.869,5.664,148.660
C00649=1211.846,75.007,-47.147,-178.872,5.664,148.661
C00650=1211.851,74.758,-47.130,-178.875,5.662,148.662
C00651=1211.856,74.509,-47.113,-178.877,5.661,148.662
C00652=1211.861,74.260,-47.096,-178.880,5.661,148.663
C00653=1211.866,74.010,-47.078,-178.882,5.660,148.663
C00654=1211.871,73.761,-47.060,-178.884,5.659,148.664
C00655=1211.875,73.512,-47.043,-178.887,5.659,148.664
C00656=1211.880,73.262,-47.026,-178.890,5.657,148.665
C00657=1211.885,73.013,-47.008,-178.892,5.657,148.666
C00658=1211.890,72.763,-46.991,-178.895,5.656,148.666
C00659=1211.895,72.514,-46.973,-178.898,5.655,148.667
C00660=1211.900,72.264,-46.956,-178.900,5.655,148.668
C00661=1211.904,72.015,-46.939,-178.902,5.654,148.668
C00662=1211.910,71.766,-46.921,-178.905,5.653,148.669
C00663=1211.914,71.517,-46.905,-178.908,5.652,148.669
C00664=1211.919,71.268,-46.887,-178.910,5.651,148.670
C00665=1211.925,71.018,-46.870,-178.913,5.650,148.670
C00666=1211.929,70.768,-46.853,-178.916,5.650,148.671
C00667=1211.934,70.519,-46.835,-178.918,5.649,148.671
C00668=1211.939,70.269,-46.818,-178.920,5.648,148.672
C00669=1211.944,70.020,-46.801,-178.923,5.648,148.673
C00670=1211.949,69.771,-46.783,-178.926,5.646,148.673
C00671=1211.954,69.522,-46.767,-178.928,5.646,148.674
C00672=1211.959,69.272,-46.749,-178.931,5.645,148.675
C00673=1211.963,69.023,-46.732,-178.934,5.644,148.675
C00674=1211.968,68.774,-46.715,-178.936,5.644,148.676
C00675=1211.973,68.524,-46.698,-178.938,5.643,148.676
C00676=1211.978,68.276,-46.681,-178.941,5.642,148.677
C00677=1211.983,68.026,-46.663,-178.944,5.641,148.678
C00678=1211.988,67.776,-46.647,-178.946,5.640,148.678
C00679=1211.993,67.527,-46.629,-178.949,5.639,148.679
C00680=1211.997,67.278,-46.612,-178.952,5.639,148.679
C00681=1212.003,67.028,-46.595,-178.954,5.638,148.680
C00682=1212.008,66.779,-46.578,-178.956,5.637,148.680
C00683=1212.013,66.529,-46.561,-178.959,5.637,148.681
C00684=1212.017,66.280,-46.544,-178.962,5.636,148.682
C00685=1212.022,66.031,-46.526,-178.964,5.636,148.682
C00686=1212.027,65.781,-46.510,-178.967,5.634,148.683
C00687=1212.033,65.532,-46.493,-178.970,5.633,148.684
C00688=1212.037,65.283,-46.476,-178.972,5.633,148.684
C00689=1212.042,65.033,-46.459,-178.974,5.632,148.685
C00690=1212.046,64.784,-46.442,-178.977,5.631,148.685
C00691=1212.052,64.535,-46.425,-178.980,5.631,148.686
C00692=1212.057,64.285,-46.408,-178.982,5.630,148.687
C00693=1212.062,64.036,-46.391,-178.984,5.629,148.687
C00694=1212.066,63.786,-46.374,-178.987,5.629,148.688
C00695=1212.072,63.537,-46.358,-178.990,5.627,148.688
C00696=1212.077,63.287,-46.340,-178.993,5.627,148.689
C00697=1212.081,63.038,-46.324,-178.995,5.626,148.689
C00698=1212.086,62.788,-46.307,-178.998,5.625,148.690
C00699=1212.091,62.540,-46.290,-179.000,5.625,148.691
C00700=1212.096,62.290,-46.272,-179.003,5.624,148.691
C00701=1212.101,62.041,-46.256,-179.005,5.623,148.692
C00702=1212.105,61.791,-46.239,-179.008,5.623,148.693
C00703=1212.111,61.542,-46.222,-179.010,5.622,148.693
C00704=1212.116,61.293,-46.205,-179.013,5.622,148.694
C00705=1212.120,61.043,-46.189,-179.016,5.620,148.694
C00706=1212.125,60.793,-46.171,-179.018,5.619,148.695
C00707=1212.130,60.545,-46.155,-179.021,5.619,148.696
C00708=1212.136,60.295,-46.138,-179.024,5.618,148.696
C00709=1212.140,60.045,-46.121,-179.026,5.617,148.697
C00710=1212.145,59.797,-46.105,-179.028,5.617,148.697
C00711=1212.150,59.547,-46.088,-179.031,5.616,148.698
C00712=1212.155,59.297,-46.071,-179.034,5.616,148.699
C00713=1212.160,59.048,-46.055,-179.036,5.615,148.699
C00714=1212.165,58.799,-46.037,-179.038,5.614,148.700
C00715=1212.170,58.549,-46.021,-179.041,5.614,148.701
C00716=1212.175,58.300,-46.004,-179.044,5.613,148.701
C00717=1212.180,58.050,-45.988,-179.046,5.612,148.702
C00718=1212.185,57.801,-45.971,-179.049,5.611,148.702
C00719=1212.190,57.552,-45.955,-179.052,5.610,148.703
C00720=1212.194,57.302,-45.938,-179.054,5.610,148.704
C00721=1212.200,57.052,-45.921,-179.056,5.609,148.704
C00722=1212.205,56.804,-45.905,-179.059,5.608,148.705
C00723=1212.209,56.554,-45.888,-179.062,5.608,148.705
C00724=1212.214,56.304,-45.871,-179.064,5.607,148.706
C00725=1212.220,56.055,-45.855,-179.067,5.607,148.707
C00726=1212.224,55.806,-45.838,-179.069,5.606,148.707
C00727=1212.229,55.538,-45.821,-179.072,5.605,148.708
C00728=1212.235,55.269,-45.802,-179.075,5.604,148.708
C00729=1212.240,55.000,-45.785,-179.078,5.603,148.709
C00730=1212.245,54.732,-45.767,-179.080,5.603,148.710
C00731=1212.250,54.483,-45.751,-179.083,5.602,148.710
C00732=1212.256,54.233,-45.734,-179.085,5.601,148.711
C00733=1212.261,53.984,-45.718,-179.088,5.601,148.712
C00734=1212.265,53.734,-45.701,-179.090,5.600,148.712
C00735=1212.270,53.485,-45.684,-179.093,5.599,148.713
C00736=1212.275,53.236,-45.668,-179.095,5.599,148.714
C00737=1212.280,52.986,-45.652,-179.098,5.598,148.714
C00738=1212.285,52.737,-45.635,-179.100,5.597,148.715
C00739=1212.290,52.487,-45.619,-179.103,5.597,148.715
C00740=1212.295,52.238,-45.603,-179.106,5.596,148.716
C00741=1212.300,51.988,-45.586,-179.109,5.595,148.717
C00742=1212.304,51.739,-45.570,-179.111,5.594,148.717
C00743=1212.310,51.490,-45.553,-179.114,5.594,148.718
C00744=1212.315,51.240,-45.537,-179.116,5.593,148.718
C00745=1212.320,50.991,-45.521,-179.119,5.592,148.719
C00746=1212.324,50.742,-45.504,-179.121,5.592,148.720
C00747=1212.330,50.492,-45.488,-179.124,5.591,148.720
C00748=1212.334,50.243,-45.472,-179.126,5.590,148.721
C00749=1212.339,49.993,-45.455,-179.129,5.590,148.722
C00750=1212.344,49.744,-45.439,-179.132,5.589,148.722
C00751=1212.349,49.494,-45.423,-179.134,5.589,148.723
C00752=1212.355,49.245,-45.406,-179.136,5.588,148.723
C00753=1212.359,48.995,-45.390,-179.139,5.587,148.724
C00754=1212.364,48.746,-45.374,-179.142,5.587,148.725
C00755=1212.369,48.496,-45.358,-179.144,5.586,148.725
C00756=1212.374,48.247,-45.341,-179.147,5.586,148.726
C00757=1212.379,47.997,-45.325,-179.149,5.585,148.726
C00758=1212.384,47.748,-45.309,-179.152,5.584,148.727
C00759=1212.389,47.499,-45.292,-179.154,5.584,148.728
C00760=1212.394,47.250,-45.277,-179.157,5.583,148.728
C00761=1212.398,47.000,-45.260,-179.160,5.583,148.729
C00762=1212.404,46.751,-45.244,-179.162,5.582,148.730
C00763=1212.408,46.501,-45.228,-179.164,5.581,148.730
C00764=1212.414,46.252,-45.212,-179.167,5.581,148.731
C00765=1212.418,46.002,-45.196,-179.170,5.580,148.732
C00766=1212.424,45.753,-45.180,-179.172,5.579,148.732
C00767=1212.428,45.503,-45.163,-179.174,5.579,148.733
C00768=1212.433,45.254,-45.148,-179.177,5.578,148.733
C00769=1212.438,45.005,-45.131,-179.180,5.577,148.734
C00770=1212.443,44.755,-45.115,-179.182,5.577,148.735
C00771=1212.448,44.506,-45.099,-179.185,5.576,148.735
C00772=1212.453,44.256,-45.083,-179.187,5.575,148.736
C00773=1212.458,44.007,-45.068,-179.190,5.575,148.737
C00774=1212.463,43.757,-45.051,-179.192,5.574,148.737
C00775=1212.468,43.508,-45.035,-179.195,5.574,148.738
C00776=1212.473,43.259,-45.019,-179.198,5.573,148.739
C00777=1212.478,43.009,-45.003,-179.200,5.572,148.739
C00778=1212.483,42.760,-44.986,-179.202,5.572,148.740
C00779=1212.488,42.510,-44.971,-179.205,5.571,148.740
C00780=1212.493,42.261,-44.955,-179.208,5.571,148.741
C00781=1212.498,42.011,-44.939,-179.210,5.570,148.742
C00782=1212.503,41.762,-44.923,-179.213,5.570,148.742
C00783=1212.508,41.512,-44.907,-179.215,5.569,148.743
C00784=1212.512,41.263,-44.891,-179.218,5.568,148.743
C00785=1212.518,41.014,-44.876,-179.220,5.568,148.744
C00786=1212.523,40.764,-44.860,-179.223,5.567,148.745
C00787=1212.528,40.515,-44.843,-179.226,5.567,148.745
C00788=1212.533,40.265,-44.828,-179.228,5.566,148.746
C00789=1212.538,40.016,-44.812,-179.230,5.565,148.747
C00790=1212.543,39.767,-44.796,-179.233,5.565,148.747
C00791=1212.548,39.517,-44.780,-179.236,5.564,148.748
C00792=1212.552,39.268,-44.765,-179.238,5.564,148.749
C00793=1212.557,39.017,-44.749,-179.241,5.563,148.749
C00794=1212.562,38.769,-44.732,-179.243,5.562,148.750
C00795=1212.568,38.519,-44.717,-179.246,5.562,148.750
C00796=1212.572,38.269,-44.701,-179.248,5.561,148.751
C00797=1212.578,38.020,-44.685,-179.251,5.560,148.752
C00798=1212.583,37.771,-44.669,-179.254,5.560,148.752
C00799=1212.587,37.521,-44.654,-179.256,5.559,148.753
C00800=1212.592,37.272,-44.638,-179.259,5.559,148.754
C00801=1212.598,37.022,-44.622,-179.261,5.558,148.754
C00802=1212.603,36.772,-44.607,-179.264,5.557,148.755
C00803=1212.608,36.524,-44.590,-179.266,5.557,148.756
C00804=1212.612,36.274,-44.575,-179.269,5.556,148.756
C00805=1212.617,36.024,-44.559,-179.272,5.556,148.757
C00806=1212.622,35.775,-44.544,-179.274,5.555,148.757
C00807=1212.628,35.526,-44.528,-179.277,5.554,148.758
C00808=1212.632,35.276,-44.513,-179.279,5.554,148.759
C00809=1212.637,35.027,-44.496,-179.282,5.553,148.759
C00810=1212.642,34.778,-44.481,-179.284,5.553,148.760
C00811=1212.647,34.527,-44.465,-179.287,5.553,148.761
C00812=1212.652,34.278,-44.450,-179.289,5.552,148.761
C00813=1212.657,34.029,-44.434,-179.291,5.552,148.762
C00814=1212.663,33.780,-44.419,-179.294,5.551,148.763
C00815=1212.667,33.529,-44.403,-179.297,5.551,148.763
C00816=1212.672,33.280,-44.388,-179.299,5.550,148.764
C00817=1212.677,33.031,-44.372,-179.302,5.549,148.765
C00818=1212.682,32.781,-44.356,-179.304,5.549,148.765
C00819=1212.686,32.532,-44.341,-179.307,5.548,148.766
C00820=1212.692,32.283,-44.325,-179.309,5.547,148.766
C00821=1212.697,32.034,-44.309,-179.312,5.547,148.767
C00822=1212.701,31.784,-44.294,-179.315,5.546,148.768
C00823=1212.707,31.534,-44.278,-179.317,5.546,148.768
C00824=1212.712,31.285,-44.263,-179.319,5.545,148.769
C00825=1212.717,31.036,-44.248,-179.322,5.544,148.770
C00826=1212.722,30.786,-44.232,-179.325,5.544,148.770
C00827=1212.727,30.536,-44.216,-179.327,5.543,148.771
C00828=1212.732,30.287,-44.201,-179.330,5.543,148.772
C00829=1212.737,30.038,-44.186,-179.333,5.542,148.772
C00830=1212.742,29.788,-44.170,-179.335,5.543,148.773
C00831=1212.747,29.519,-44.154,-179.338,5.541,148.774
C00832=1212.752,29.251,-44.137,-179.341,5.541,148.774
C00833=1212.758,28.981,-44.121,-179.343,5.540,148.775
C00834=1212.763,28.713,-44.104,-179.346,5.540,148.776
C00835=1212.768,28.464,-44.089,-179.349,5.539,148.776
C00836=1212.774,28.214,-44.073,-179.351,5.539,148.777
C00837=1212.778,27.965,-44.058,-179.353,5.538,148.777
C00838=1212.783,27.715,-44.042,-179.356,5.537,148.778
C00839=1212.788,27.466,-44.027,-179.358,5.537,148.779
C00840=1212.794,27.216,-44.012,-179.361,5.537,148.780
C00841=1212.799,26.967,-43.997,-179.363,5.536,148.780
C00842=1212.804,26.718,-43.982,-179.366,5.536,148.781
C00843=1212.808,26.468,-43.966,-179.369,5.535,148.782
C00844=1212.813,26.218,-43.951,-179.371,5.534,148.782
C00845=1212.819,25.969,-43.935,-179.373,5.534,148.783
C00846=1212.823,25.720,-43.920,-179.376,5.533,148.783
C00847=1212.829,25.470,-43.905,-179.379,5.533,148.784
C00848=1212.833,25.220,-43.890,-179.381,5.532,148.785
C00849=1212.838,24.971,-43.874,-179.384,5.532,148.785
C00850=1212.843,24.722,-43.859,-179.387,5.531,148.786
C00851=1212.848,24.472,-43.844,-179.388,5.531,148.787
C00852=1212.853,24.223,-43.830,-179.391,5.531,148.787
C00853=1212.859,23.973,-43.814,-179.394,5.530,148.788
C00854=1212.863,23.724,-43.799,-179.396,5.530,148.789
C00855=1212.868,23.474,-43.783,-179.399,5.529,148.789
C00856=1212.873,23.224,-43.769,-179.401,5.529,148.790
C00857=1212.878,22.975,-43.753,-179.404,5.528,148.791
C00858=1212.883,22.726,-43.738,-179.407,5.528,148.791
C00859=1212.888,22.476,-43.723,-179.409,5.527,148.792
C00860=1212.893,22.227,-43.708,-179.412,5.526,148.792
C00861=1212.899,21.977,-43.693,-179.414,5.526,148.793
C00862=1212.903,21.728,-43.678,-179.416,5.526,148.794
C00863=1212.909,21.477,-43.662,-179.419,5.525,148.794
C00864=1212.913,21.228,-43.647,-179.422,5.525,148.795
C00865=1212.918,20.979,-43.632,-179.424,5.524,148.796
C00866=1212.924,20.729,-43.618,-179.426,5.523,148.796
C00867=1212.928,20.480,-43.603,-179.429,5.523,148.797
C00868=1212.934,20.231,-43.587,-179.432,5.522,148.798
C00869=1212.939,19.981,-43.573,-179.434,5.522,148.798
C00870=1212.943,19.732,-43.558,-179.437,5.521,148.799
C00871=1212.949,19.482,-43.542,-179.439,5.522,148.800
C00872=1212.954,19.233,-43.528,-179.442,5.521,148.800
C00873=1212.959,18.983,-43.512,-179.444,5.521,148.801
C00874=1212.964,18.734,-43.498,-179.446,5.520,148.801
C00875=1212.969,18.485,-43.483,-179.449,5.519,148.802
C00876=1212.973,18.234,-43.467,-179.452,5.519,148.803
C00877=1212.978,17.985,-43.453,-179.454,5.518,148.804
C00878=1212.983,17.736,-43.438,-179.457,5.518,148.804
C00879=1212.989,17.486,-43.423,-179.460,5.517,148.805
C00880=1212.993,17.237,-43.408,-179.462,5.517,148.806
C00881=1212.998,16.987,-43.394,-179.464,5.517,148.806
C00882=1213.004,16.737,-43.378,-179.467,5.516,148.807
C00883=1213.009,16.488,-43.364,-179.469,5.515,148.807
C00884=1213.013,16.239,-43.349,-179.472,5.515,148.808
C00885=1213.019,15.989,-43.334,-179.475,5.514,148.809
C00886=1213.024,15.740,-43.319,-179.477,5.514,148.809
C00887=1213.028,15.490,-43.305,-179.480,5.513,148.810
C00888=1213.034,15.240,-43.289,-179.482,5.514,148.811
C00889=1213.039,14.991,-43.275,-179.485,5.513,148.812
C00890=1213.043,14.742,-43.260,-179.487,5.513,148.812
C00891=1213.049,14.492,-43.245,-179.489,5.512,148.813
C00892=1213.054,14.243,-43.230,-179.492,5.511,148.813
C00893=1213.059,13.993,-43.216,-179.495,5.511,148.814
C00894=1213.063,13.744,-43.201,-179.497,5.510,148.815
C00895=1213.069,13.494,-43.186,-179.499,5.510,148.815
C00896=1213.074,13.245,-43.171,-179.502,5.510,148.816
C00897=1213.079,12.995,-43.157,-179.505,5.509,148.817
C00898=1213.084,12.745,-43.142,-179.507,5.509,148.817
C00899=1213.089,12.496,-43.127,-179.510,5.508,148.818
C00900=1213.094,12.246,-43.112,-179.512,5.507,148.819
C00901=1213.099,11.996,-43.098,-179.515,5.507,148.819
C00902=1213.104,11.747,-43.083,-179.517,5.507,148.820
C00903=1213.109,11.497,-43.068,-179.520,5.507,148.821
C00904=1213.114,11.248,-43.053,-179.522,5.506,148.821
C00905=1213.119,10.998,-43.039,-179.525,5.506,148.822
C00906=1213.124,10.749,-43.025,-179.527,5.505,148.823
C00907=1213.129,10.500,-43.010,-179.530,5.505,148.823
C00908=1213.135,10.250,-42.995,-179.533,5.504,148.824
C00909=1213.140,10.001,-42.981,-179.534,5.504,148.825
C00910=1213.144,9.752,-42.966,-179.537,5.504,148.825
C00911=1213.149,9.502,-42.952,-179.540,5.503,148.826
C00912=1213.154,9.252,-42.937,-179.542,5.503,148.827
C00913=1213.159,9.002,-42.923,-179.545,5.502,148.827
C00914=1213.164,8.753,-42.908,-179.548,5.501,148.828
C00915=1213.170,8.503,-42.893,-179.550,5.502,148.829
C00916=1213.175,8.254,-42.879,-179.552,5.501,148.829
C00917=1213.180,8.004,-42.865,-179.555,5.501,148.830
C00918=1213.184,7.755,-42.850,-179.558,5.500,148.831
C00919=1213.190,7.506,-42.836,-179.560,5.499,148.831
C00920=1213.195,7.256,-42.821,-179.562,5.499,148.832
C00921=1213.200,7.006,-42.807,-179.565,5.498,148.833
C00922=1213.204,6.757,-42.792,-179.567,5.499,148.833
C00923=1213.210,6.507,-42.777,-179.570,5.498,148.834
C00924=1213.215,6.257,-42.763,-179.572,5.498,148.835
C00925=1213.220,6.008,-42.749,-179.575,5.497,148.835
C00926=1213.225,5.758,-42.735,-179.578,5.497,148.836
C00927=1213.230,5.510,-42.720,-179.580,5.496,148.837
C00928=1213.235,5.260,-42.706,-179.582,5.496,148.837
C00929=1213.240,5.010,-42.691,-179.585,5.495,148.838
C00930=1213.245,4.761,-42.677,-179.587,5.495,148.838
C00931=1213.250,4.511,-42.663,-179.590,5.494,148.839
C00932=1213.255,4.261,-42.649,-179.593,5.494,148.840
C00933=1213.260,4.011,-42.634,-179.595,5.494,148.841
C00934=1213.265,3.763,-42.620,-179.597,5.494,148.841
C00935=1213.271,3.494,-42.605,-179.600,5.493,148.842
C00936=1213.276,3.225,-42.588,-179.603,5.493,148.843
C00937=1213.282,2.955,-42.573,-179.605,5.492,148.843
C00938=1213.287,2.686,-42.558,-179.608,5.492,148.844
C00939=1213.292,2.437,-42.543,-179.611,5.491,148.845
C00940=1213.297,2.187,-42.529,-179.613,5.491,148.845
C00941=1213.302,1.938,-42.515,-179.616,5.490,148.846
C00942=1213.307,1.688,-42.501,-179.618,5.490,148.847
C00943=1213.312,1.438,-42.487,-179.621,5.490,148.847
C00944=1213.317,1.189,-42.472,-179.623,5.489,148.848
C00945=1213.322,0.939,-42.458,-179.626,5.489,148.849
C00946=1213.328,0.690,-42.444,-179.629,5.488,148.849
C00947=1213.333,0.440,-42.430,-179.631,5.489,148.850
C00948=1213.338,0.191,-42.416,-179.633,5.488,148.851
C00949=1213.343,-0.059,-42.401,-179.635,5.487,148.851
C00950=1213.348,-0.308,-42.387,-179.638,5.487,148.852
C00951=1213.353,-0.558,-42.373,-179.641,5.486,148.853
C00952=1213.357,-0.807,-42.359,-179.643,5.487,148.853
C00953=1213.362,-1.057,-42.345,-179.646,5.486,148.854
C00954=1213.367,-1.307,-42.331,-179.648,5.486,148.855
C00955=1213.373,-1.556,-42.317,-179.651,5.485,148.855
C00956=1213.378,-1.805,-42.303,-179.653,5.485,148.856
C00957=1213.383,-2.055,-42.288,-179.656,5.485,148.857
C00958=1213.388,-2.305,-42.274,-179.658,5.484,148.858
C00959=1213.393,-2.554,-42.260,-179.661,5.484,148.858
C00960=1213.398,-2.804,-42.246,-179.663,5.483,148.859
C00961=1213.403,-3.053,-42.232,-179.666,5.483,148.859
C00962=1213.408,-3.304,-42.218,-179.668,5.483,148.860
C00963=1213.413,-3.552,-42.205,-179.670,5.482,148.861
C00964=1213.418,-3.802,-42.190,-179.673,5.482,148.861
C00965=1213.423,-4.052,-42.176,-179.676,5.481,148.862
C00966=1213.429,-4.301,-42.162,-179.678,5.481,148.863
C00967=1213.434,-4.550,-42.148,-179.680,5.481,148.863
C00968=1213.439,-4.800,-42.134,-179.683,5.481,148.864
C00969=1213.444,-5.050,-42.120,-179.686,5.480,148.865
C00970=1213.449,-5.299,-42.107,-179.688,5.480,148.866
C00971=1213.454,-5.549,-42.093,-179.691,5.479,148.866
C00972=1213.459,-5.799,-42.078,-179.693,5.479,148.867
C00973=1213.464,-6.048,-42.064,-179.695,5.479,148.867
C00974=1213.469,-6.297,-42.050,-179.698,5.478,148.868
C00975=1213.474,-6.547,-42.037,-179.701,5.478,148.869
C00976=1213.479,-6.796,-42.023,-179.703,5.478,148.869
C00977=1213.484,-7.046,-42.009,-179.705,5.477,148.870
C00978=1213.489,-7.296,-41.995,-179.708,5.477,148.871
C00979=1213.494,-7.546,-41.981,-179.711,5.476,148.872
C00980=1213.499,-7.795,-41.968,-179.713,5.476,148.872
C00981=1213.504,-8.044,-41.954,-179.715,5.476,148.873
C00982=1213.509,-8.294,-41.939,-179.718,5.476,148.874
C00983=1213.515,-8.544,-41.926,-179.721,5.475,148.874
C00984=1213.519,-8.793,-41.912,-179.723,5.475,148.875
C00985=1213.524,-9.043,-41.898,-179.725,5.475,148.875
C00986=1213.530,-9.292,-41.884,-179.728,5.474,148.876
C00987=1213.535,-9.542,-41.871,-179.730,5.474,148.877
C00988=1213.540,-9.791,-41.857,-179.733,5.473,148.878
C00989=1213.545,-10.041,-41.843,-179.735,5.473,148.878
C00990=1213.550,-10.291,-41.829,-179.738,5.473,148.879
C00991=1213.556,-10.540,-41.816,-179.740,5.472,148.880
C00992=1213.560,-10.789,-41.802,-179.743,5.472,148.880
C00993=1213.565,-11.040,-41.788,-179.746,5.471,148.881
C00994=1213.571,-11.289,-41.774,-179.748,5.472,148.882
C00995=1213.575,-11.538,-41.761,-179.750,5.471,148.882
C00996=1213.581,-11.788,-41.748,-179.753,5.471,148.883
C00997=1213.586,-12.037,-41.733,-179.756,5.470,148.884
C00998=1213.590,-12.287,-41.720,-179.757,5.470,148.884
C00999=1213.596,-12.536,-41.706,-179.760,5.470,148.885
C01000=1213.601,-12.786,-41.692,-179.763,5.469,148.886
C01001=1213.605,-13.036,-41.679,-179.765,5.469,148.886
C01002=1213.611,-13.285,-41.665,-179.767,5.469,148.887
C01003=1213.616,-13.536,-41.652,-179.770,5.469,148.888
C01004=1213.621,-13.784,-41.638,-179.773,5.468,148.888
C01005=1213.626,-14.034,-41.624,-179.775,5.468,148.889
C01006=1213.632,-14.284,-41.611,-179.777,5.468,148.890
C01007=1213.636,-14.533,-41.597,-179.780,5.467,148.890
C01008=1213.641,-14.783,-41.584,-179.783,5.467,148.891
C01009=1213.647,-15.032,-41.570,-179.785,5.466,148.892
C01010=1213.651,-15.282,-41.557,-179.787,5.467,148.893
C01011=1213.657,-15.531,-41.543,-179.790,5.466,148.893
C01012=1213.661,-15.781,-41.530,-179.792,5.465,148.894
C01013=1213.667,-16.030,-41.516,-179.795,5.465,148.894
C01014=1213.672,-16.281,-41.502,-179.797,5.465,148.895
C01015=1213.677,-16.529,-41.489,-179.800,5.465,148.896
C01016=1213.682,-16.780,-41.476,-179.802,5.464,148.896
C01017=1213.686,-17.029,-41.462,-179.805,5.464,148.897
C01018=1213.692,-17.279,-41.449,-179.807,5.464,148.898
C01019=1213.697,-17.528,-41.434,-179.810,5.463,148.899
C01020=1213.702,-17.778,-41.422,-179.812,5.463,148.899
C01021=1213.707,-18.028,-41.407,-179.814,5.463,148.900
C01022=1213.712,-18.277,-41.395,-179.817,5.463,148.901
C01023=1213.718,-18.527,-41.381,-179.820,5.462,148.901
C01024=1213.722,-18.776,-41.368,-179.822,5.462,148.902
C01025=1213.728,-19.026,-41.354,-179.824,5.462,148.903
C01026=1213.733,-19.275,-41.341,-179.827,5.461,148.903
C01027=1213.738,-19.525,-41.328,-179.829,5.461,148.904
C01028=1213.743,-19.775,-41.315,-179.832,5.460,148.905
C01029=1213.748,-20.024,-41.301,-179.834,5.461,148.905
C01030=1213.754,-20.274,-41.288,-179.837,5.460,148.906
C01031=1213.758,-20.524,-41.275,-179.839,5.460,148.907
C01032=1213.764,-20.773,-41.261,-179.842,5.459,148.907
C01033=1213.768,-21.023,-41.248,-179.844,5.459,148.908
C01034=1213.774,-21.273,-41.234,-179.847,5.459,148.909
C01035=1213.778,-21.522,-41.221,-179.849,5.458,148.909
C01036=1213.784,-21.771,-41.208,-179.851,5.459,148.910
C01037=1213.789,-22.021,-41.195,-179.854,5.458,148.911
C01038=1213.794,-22.270,-41.181,-179.857,5.458,148.912
C01039=1213.799,-22.540,-41.167,-179.859,5.457,148.912
C01040=1213.805,-22.809,-41.152,-179.862,5.457,148.913
C01041=1213.810,-23.079,-41.139,-179.864,5.457,148.914
C01042=1213.816,-23.348,-41.124,-179.867,5.457,148.914
C01043=1213.821,-23.598,-41.111,-179.870,5.456,148.915
C01044=1213.826,-23.848,-41.098,-179.872,5.456,148.916
C01045=1213.831,-24.097,-41.085,-179.874,5.456,148.916
C01046=1213.836,-24.347,-41.071,-179.877,5.456,148.917
C01047=1213.841,-24.596,-41.058,-179.880,5.455,148.918
C01048=1213.847,-24.846,-41.045,-179.882,5.455,148.919
C01049=1213.852,-25.096,-41.032,-179.884,5.455,148.919
C01050=1213.857,-25.345,-41.019,-179.887,5.454,148.920
C01051=1213.862,-25.595,-41.005,-179.890,5.454,148.921
C01052=1213.867,-25.844,-40.992,-179.892,5.454,148.921
C01053=1213.872,-26.094,-40.979,-179.894,5.453,148.922
C01054=1213.877,-26.344,-40.966,-179.897,5.453,148.922
C01055=1213.882,-26.593,-40.953,-179.899,5.453,148.923
C01056=1213.887,-26.843,-40.939,-179.901,5.453,148.924
C01057=1213.893,-27.092,-40.927,-179.904,5.452,148.925
C01058=1213.897,-27.342,-40.914,-179.907,5.452,148.925
C01059=1213.903,-27.592,-40.901,-179.909,5.452,148.926
C01060=1213.908,-27.841,-40.888,-179.911,5.452,148.927
C01061=1213.913,-28.091,-40.875,-179.914,5.451,148.927
C01062=1213.918,-28.340,-40.861,-179.916,5.451,148.928
C01063=1213.923,-28.589,-40.849,-179.919,5.451,148.929
C01064=1213.928,-28.840,-40.836,-179.921,5.450,148.929
C01065=1213.934,-29.089,-40.822,-179.923,5.451,148.930
C01066=1213.938,-29.339,-40.809,-179.926,5.450,148.931
C01067=1213.943,-29.588,-40.797,-179.929,5.450,148.932
C01068=1213.948,-29.838,-40.784,-179.931,5.449,148.932
C01069=1213.954,-30.088,-40.771,-179.933,5.449,148.933
C01070=1213.959,-30.337,-40.758,-179.936,5.449,148.933
C01071=1213.964,-30.587,-40.745,-179.938,5.448,148.934
C01072=1213.969,-30.837,-40.732,-179.940,5.449,148.935
C01073=1213.974,-31.086,-40.719,-179.943,5.448,148.935
C01074=1213.979,-31.336,-40.707,-179.946,5.448,148.936
C01075=1213.984,-31.585,-40.693,-179.948,5.448,148.937
C01076=1213.990,-31.835,-40.680,-179.951,5.448,148.938
C01077=1213.995,-32.084,-40.667,-179.953,5.447,148.938
C01078=1213.999,-32.334,-40.654,-179.955,5.447,148.939
C01079=1214.004,-32.583,-40.642,-179.958,5.447,148.940
C01080=1214.010,-32.833,-40.628,-179.961,5.446,148.940
C01081=1214.015,-33.083,-40.616,-179.963,5.446,148.941
C01082=1214.020,-33.333,-40.604,-179.965,5.446,148.942
C01083=1214.025,-33.582,-40.591,-179.967,5.445,148.942
C01084=1214.031,-33.832,-40.578,-179.970,5.445,148.943
C01085=1214.036,-34.082,-40.565,-179.972,5.445,148.944
C01086=1214.041,-34.331,-40.552,-179.975,5.445,148.944
C01087=1214.046,-34.581,-40.540,-179.978,5.444,148.945
C01088=1214.050,-34.831,-40.527,-179.980,5.445,148.946
C01089=1214.056,-35.080,-40.513,-179.982,5.444,148.946
C01090=1214.061,-35.330,-40.501,-179.985,5.444,148.947
C01091=1214.067,-35.579,-40.488,-179.987,5.444,148.948
C01092=1214.071,-35.829,-40.475,-179.990,5.444,148.949
C01093=1214.076,-36.078,-40.463,-179.992,5.443,148.949
C01094=1214.082,-36.328,-40.450,-179.994,5.443,148.950
C01095=1214.087,-36.578,-40.438,-179.997,5.443,148.951
C01096=1214.092,-36.828,-40.425,-180.000,5.442,148.951
C01097=1214.097,-37.077,-40.412,179.998,5.443,148.952
C01098=1214.102,-37.326,-40.399,179.996,5.442,148.952
C01099=1214.107,-37.576,-40.387,179.993,5.441,148.953
C01100=1214.112,-37.826,-40.374,179.991,5.442,148.954
C01101=1214.118,-38.075,-40.361,179.989,5.441,148.955
C01102=1214.123,-38.325,-40.349,179.986,5.441,148.955
C01103=1214.128,-38.575,-40.336,179.984,5.441,148.956
C01104=1214.133,-38.825,-40.323,179.981,5.441,148.957
C01105=1214.138,-39.074,-40.311,179.978,5.440,148.957
C01106=1214.143,-39.323,-40.298,179.976,5.441,148.958
C01107=1214.148,-39.573,-40.286,179.974,5.440,148.959
C01108=1214.154,-39.823,-40.274,179.971,5.440,148.959
C01109=1214.158,-40.073,-40.261,179.969,5.440,148.960
C01110=1214.163,-40.322,-40.248,179.966,5.439,148.961
C01111=1214.169,-40.572,-40.236,179.964,5.439,148.962
C01112=1214.175,-40.821,-40.223,179.962,5.439,148.962
C01113=1214.180,-41.071,-40.210,179.959,5.438,148.963
C01114=1214.184,-41.321,-40.197,179.957,5.438,148.963
C01115=1214.190,-41.571,-40.185,179.955,5.438,148.964
C01116=1214.195,-41.820,-40.173,179.952,5.438,148.965
C01117=1214.200,-42.069,-40.160,179.950,5.438,148.966
C01118=1214.205,-42.319,-40.148,179.947,5.438,148.966
C01119=1214.210,-42.569,-40.135,179.945,5.437,148.967
C01120=1214.215,-42.819,-40.123,179.943,5.438,148.968
C01121=1214.220,-43.068,-40.110,179.940,5.437,148.968
C01122=1214.226,-43.318,-40.098,179.937,5.437,148.969
C01123=1214.231,-43.567,-40.086,179.935,5.437,148.970
C01124=1214.236,-43.817,-40.073,179.932,5.436,148.970
C01125=1214.241,-44.067,-40.061,179.930,5.436,148.971
C01126=1214.246,-44.316,-40.048,179.928,5.436,148.972
C01127=1214.251,-44.566,-40.036,179.926,5.436,148.972
C01128=1214.256,-44.816,-40.024,179.923,5.435,148.973
C01129=1214.261,-45.065,-40.011,179.921,5.435,148.974
C01130=1214.267,-45.314,-39.999,179.918,5.435,148.974
C01131=1214.272,-45.564,-39.987,179.915,5.434,148.975
C01132=1214.277,-45.814,-39.974,179.913,5.435,148.976
C01133=1214.282,-46.064,-39.962,179.911,5.434,148.977
C01134=1214.287,-46.314,-39.949,179.909,5.435,148.977
C01135=1214.292,-46.564,-39.937,179.906,5.434,148.978
C01136=1214.298,-46.813,-39.925,179.903,5.434,148.979
C01137=1214.303,-47.062,-39.912,179.901,5.434,148.979
C01138=1214.308,-47.312,-39.900,179.899,5.434,148.980
C01139=1214.313,-47.561,-39.888,179.896,5.433,148.981
C01140=1214.318,-47.811,-39.876,179.894,5.433,148.981
C01141=1214.323,-48.060,-39.864,179.892,5.433,148.982
C01142=1214.328,-48.311,-39.852,179.889,5.432,148.983
C01143=1214.333,-48.580,-39.838,179.886,5.433,148.984
C01144=1214.340,-48.851,-39.825,179.884,5.432,148.984
C01145=1214.345,-49.121,-39.812,179.881,5.432,148.985
C01146=1214.350,-49.390,-39.798,179.878,5.431,148.986
C01147=1214.356,-49.640,-39.786,179.876,5.432,148.986
C01148=1214.361,-49.889,-39.774,179.874,5.431,148.987
C01149=1214.366,-50.139,-39.762,179.872,5.432,148.988
C01150=1214.372,-50.389,-39.749,179.869,5.431,148.989
C01151=1214.376,-50.638,-39.738,179.866,5.431,148.989
C01152=1214.381,-50.888,-39.725,179.864,5.431,148.990
C01153=1214.386,-51.138,-39.713,179.861,5.431,148.991
C01154=1214.391,-51.387,-39.701,179.859,5.430,148.991
C01155=1214.397,-51.637,-39.689,179.857,5.430,148.992
C01156=1214.402,-51.887,-39.677,179.855,5.430,148.992
C01157=1214.407,-52.136,-39.665,179.852,5.430,148.993
C01158=1214.412,-52.386,-39.653,179.850,5.430,148.994
C01159=1214.417,-52.636,-39.640,179.847,5.429,148.995
C01160=1214.423,-52.886,-39.629,179.845,5.429,148.995
C01161=1214.428,-53.135,-39.617,179.842,5.429,148.996
C01162=1214.433,-53.385,-39.604,179.840,5.428,148.997
C01163=1214.438,-53.634,-39.593,179.838,5.429,148.997
C01164=1214.443,-53.884,-39.580,179.835,5.428,148.998
C01165=1214.448,-54.134,-39.568,179.833,5.429,148.999
C01166=1214.454,-54.384,-39.556,179.830,5.428,149.000
C01167=1214.458,-54.633,-39.544,179.828,5.427,149.000
C01168=1214.464,-54.883,-39.532,179.826,5.428,149.001
C01169=1214.469,-55.132,-39.521,179.823,5.427,149.001
C01170=1214.474,-55.382,-39.508,179.821,5.428,149.002
C01171=1214.479,-55.631,-39.497,179.818,5.427,149.003
C01172=1214.484,-55.881,-39.485,179.816,5.427,149.004
C01173=1214.489,-56.131,-39.472,179.814,5.427,149.004
C01174=1214.495,-56.381,-39.460,179.811,5.427,149.005
C01175=1214.500,-56.630,-39.449,179.809,5.427,149.006
C01176=1214.505,-56.880,-39.437,179.806,5.426,149.006
C01177=1214.510,-57.129,-39.425,179.804,5.426,149.007
C01178=1214.515,-57.379,-39.413,179.802,5.426,149.008
C01179=1214.520,-57.629,-39.401,179.799,5.426,149.008
C01180=1214.525,-57.878,-39.389,179.797,5.425,149.009
C01181=1214.531,-58.128,-39.377,179.795,5.425,149.010
C01182=1214.535,-58.378,-39.366,179.792,5.425,149.010
C01183=1214.541,-58.628,-39.354,179.790,5.425,149.011
C01184=1214.546,-58.878,-39.342,179.787,5.425,149.012
C01185=1214.551,-59.127,-39.330,179.785,5.424,149.012
C01186=1214.556,-59.377,-39.318,179.782,5.425,149.013
C01187=1214.562,-59.627,-39.306,179.780,5.424,149.014
C01188=1214.566,-59.876,-39.295,179.778,5.425,149.015
C01189=1214.571,-60.126,-39.282,179.775,5.424,149.015
C01190=1214.577,-60.375,-39.271,179.773,5.424,149.016
C01191=1214.582,-60.624,-39.259,179.770,5.424,149.017
C01192=1214.588,-60.874,-39.247,179.768,5.423,149.017
C01193=1214.593,-61.124,-39.236,179.766,5.424,149.018
C01194=1214.598,-61.374,-39.224,179.763,5.423,149.019
C01195=1214.603,-61.624,-39.212,179.761,5.423,149.019
C01196=1214.608,-61.873,-39.200,179.759,5.423,149.020
C01197=1214.613,-62.123,-39.189,179.756,5.423,149.021
C01198=1214.618,-62.373,-39.177,179.754,5.423,149.021
C01199=1214.623,-62.622,-39.165,179.751,5.422,149.022
C01200=1214.628,-62.872,-39.153,179.749,5.423,149.023
C01201=1214.634,-63.122,-39.142,179.746,5.422,149.024
C01202=1214.639,-63.371,-39.131,179.744,5.422,149.024
C01203=1214.645,-63.621,-39.119,179.742,5.422,149.025
C01204=1214.649,-63.871,-39.107,179.740,5.421,149.025
C01205=1214.654,-64.120,-39.095,179.737,5.422,149.026
C01206=1214.660,-64.370,-39.083,179.735,5.421,149.027
C01207=1214.665,-64.620,-39.072,179.732,5.421,149.028
C01208=1214.670,-64.870,-39.060,179.730,5.421,149.028
C01209=1214.675,-65.119,-39.049,179.727,5.421,149.029
C01210=1214.681,-65.368,-39.037,179.725,5.421,149.030
C01211=1214.685,-65.618,-39.026,179.723,5.421,149.030
C01212=1214.691,-65.868,-39.014,179.720,5.421,149.031
C01213=1214.696,-66.118,-39.002,179.718,5.421,149.032
C01214=1214.701,-66.368,-38.991,179.715,5.420,149.032
C01215=1214.706,-66.618,-38.979,179.714,5.420,149.033
C01216=1214.712,-66.866,-38.968,179.711,5.420,149.034
C01217=1214.717,-67.116,-38.956,179.709,5.420,149.034
C01218=1214.722,-67.366,-38.945,179.706,5.419,149.035
C01219=1214.727,-67.616,-38.933,179.704,5.420,149.036
C01220=1214.732,-67.866,-38.921,179.701,5.419,149.036
C01221=1214.737,-68.116,-38.910,179.699,5.419,149.037
C01222=1214.743,-68.364,-38.899,179.697,5.419,149.038
C01223=1214.748,-68.614,-38.887,179.694,5.419,149.039
C01224=1214.753,-68.864,-38.876,179.692,5.419,149.039
C01225=1214.758,-69.114,-38.864,179.690,5.418,149.040
C01226=1214.763,-69.364,-38.853,179.688,5.419,149.040
C01227=1214.769,-69.613,-38.842,179.685,5.418,149.041
C01228=1214.774,-69.863,-38.830,179.682,5.418,149.042
C01229=1214.779,-70.113,-38.818,179.680,5.418,149.043
C01230=1214.784,-70.363,-38.807,179.677,5.418,149.043
C01231=1214.789,-70.612,-38.796,179.675,5.418,149.044
C01232=1214.795,-70.861,-38.784,179.673,5.418,149.045
C01233=1214.799,-71.111,-38.773,179.671,5.418,149.045
C01234=1214.805,-71.361,-38.761,179.668,5.418,149.046
C01235=1214.810,-71.611,-38.751,179.666,5.417,149.047
C01236=1214.816,-71.861,-38.739,179.664,5.417,149.047
C01237=1214.821,-72.110,-38.728,179.661,5.417,149.048
C01238=1214.826,-72.360,-38.716,179.659,5.417,149.049
C01239=1214.831,-72.610,-38.705,179.656,5.417,149.049
C01240=1214.836,-72.859,-38.694,179.654,5.417,149.050
C01241=1214.841,-73.109,-38.682,179.652,5.416,149.051
C01242=1214.846,-73.359,-38.671,179.649,5.416,149.052
C01243=1214.852,-73.609,-38.659,179.647,5.416,149.052
C01244=1214.857,-73.858,-38.648,179.644,5.416,149.053
C01245=1214.862,-74.107,-38.637,179.643,5.416,149.053
C01246=1214.868,-74.358,-38.626,179.640,5.415,149.054
C01247=1214.873,-74.628,-38.613,179.638,5.416,149.055
C01248=1214.878,-74.898,-38.602,179.635,5.416,149.056
C01249=1214.884,-75.169,-38.589,179.632,5.415,149.057
C01250=1214.890,-75.439,-38.577,179.630,5.416,149.057
C01251=1214.895,-75.689,-38.566,179.627,5.415,149.058
C01252=1214.900,-75.939,-38.554,179.624,5.415,149.059
C01253=1214.905,-76.189,-38.543,179.622,5.415,149.059
C01254=1214.911,-76.438,-38.532,179.620,5.414,149.060
C01255=1214.916,-76.688,-38.521,179.618,5.415,149.061
C01256=1214.921,-76.938,-38.510,179.615,5.414,149.061
C01257=1214.927,-77.188,-38.499,179.613,5.415,149.062
C01258=1214.932,-77.437,-38.488,179.611,5.414,149.063
C01259=1214.936,-77.687,-38.476,179.609,5.414,149.063
C01260=1214.942,-77.936,-38.465,179.606,5.414,149.064
C01261=1214.947,-78.186,-38.454,179.603,5.414,149.065
C01262=1214.952,-78.436,-38.443,179.601,5.414,149.066
C01263=1214.957,-78.685,-38.432,179.599,5.413,149.066
C01264=1214.963,-78.935,-38.421,179.597,5.413,149.067
C01265=1214.968,-79.185,-38.409,179.594,5.413,149.067
C01266=1214.973,-79.434,-38.399,179.592,5.413,149.068
C01267=1214.978,-79.684,-38.388,179.589,5.413,149.069
C01268=1214.984,-79.934,-38.376,179.587,5.413,149.070
C01269=1214.989,-80.184,-38.366,179.585,5.413,149.070
C01270=1214.994,-80.433,-38.355,179.583,5.413,149.071
C01271=1214.999,-80.683,-38.343,179.580,5.412,149.071
C01272=1215.005,-80.933,-38.333,179.578,5.412,149.072
C01273=1215.010,-81.182,-38.321,179.576,5.412,149.073
C01274=1215.015,-81.433,-38.311,179.573,5.412,149.074
C01275=1215.020,-81.682,-38.300,179.571,5.412,149.074
C01276=1215.025,-81.932,-38.288,179.568,5.412,149.075
C01277=1215.030,-82.182,-38.277,179.566,5.412,149.076
C01278=1215.036,-82.431,-38.266,179.563,5.412,149.076
C01279=1215.041,-82.681,-38.256,179.562,5.412,149.077
C01280=1215.045,-82.931,-38.244,179.559,5.411,149.078
C01281=1215.052,-83.180,-38.234,179.557,5.412,149.078
C01282=1215.056,-83.430,-38.222,179.554,5.411,149.079
C01283=1215.062,-83.680,-38.212,179.552,5.412,149.080
C01284=1215.067,-83.929,-38.201,179.550,5.411,149.080
C01285=1215.072,-84.179,-38.190,179.547,5.411,149.081
C01286=1215.078,-84.429,-38.179,179.545,5.411,149.082
C01287=1215.083,-84.679,-38.168,179.543,5.410,149.082
C01288=1215.088,-84.928,-38.157,179.541,5.411,149.083
C01289=1215.093,-85.178,-38.147,179.538,5.410,149.084
C01290=1215.098,-85.428,-38.135,179.536,5.410,149.084
C01291=1215.103,-85.677,-38.125,179.533,5.410,149.085
C01292=1215.108,-85.927,-38.114,179.531,5.410,149.086
C01293=1215.114,-86.177,-38.103,179.528,5.410,149.087
C01294=1215.119,-86.426,-38.092,179.526,5.410,149.087
C01295=1215.124,-86.677,-38.081,179.524,5.410,149.088
C01296=1215.129,-86.926,-38.070,179.522,5.410,149.089
C01297=1215.134,-87.176,-38.060,179.519,5.409,149.089
C01298=1215.140,-87.425,-38.050,179.517,5.410,149.090
C01299=1215.144,-87.675,-38.038,179.515,5.409,149.091
C01300=1215.150,-87.925,-38.028,179.513,5.410,149.091
C01301=1215.155,-88.174,-38.017,179.510,5.409,149.092
C01302=1215.161,-88.424,-38.006,179.508,5.409,149.093
C01303=1215.166,-88.674,-37.995,179.506,5.409,149.093
C01304=1215.171,-88.924,-37.984,179.503,5.408,149.094
C01305=1215.176,-89.173,-37.974,179.501,5.409,149.095
C01306=1215.181,-89.423,-37.963,179.498,5.408,149.095
C01307=1215.187,-89.673,-37.952,179.496,5.409,149.096
C01308=1215.192,-89.923,-37.942,179.493,5.408,149.097
C01309=1215.197,-90.172,-37.931,179.492,5.408,149.097
C01310=1215.202,-90.422,-37.920,179.489,5.408,149.098
C01311=1215.208,-90.672,-37.910,179.487,5.408,149.099
C01312=1215.212,-90.921,-37.899,179.484,5.408,149.099
C01313=1215.218,-91.171,-37.889,179.482,5.408,149.100
C01314=1215.223,-91.421,-37.878,179.480,5.408,149.101
C01315=1215.228,-91.670,-37.867,179.478,5.408,149.102
C01316=1215.233,-91.920,-37.857,179.475,5.407,149.102
C01317=1215.239,-92.170,-37.846,179.473,5.408,149.103
C01318=1215.244,-92.420,-37.836,179.471,5.407,149.103
C01319=1215.249,-92.669,-37.825,179.469,5.408,149.104
C01320=1215.254,-92.919,-37.814,179.466,5.407,149.105
C01321=1215.260,-93.169,-37.804,179.464,5.408,149.106
C01322=1215.264,-93.418,-37.793,179.461,5.407,149.106
C01323=1215.270,-93.668,-37.783,179.460,5.407,149.107
C01324=1215.275,-93.918,-37.772,179.457,5.407,149.108
C01325=1215.281,-94.168,-37.762,179.455,5.407,149.108
C01326=1215.286,-94.418,-37.751,179.452,5.407,149.109
C01327=1215.291,-94.667,-37.740,179.450,5.407,149.110
C01328=1215.296,-94.917,-37.730,179.447,5.407,149.110
C01329=1215.301,-95.167,-37.719,179.446,5.407,149.111
C01330=1215.307,-95.416,-37.709,179.443,5.406,149.112
C01331=1215.312,-95.666,-37.698,179.441,5.406,149.112
C01332=1215.317,-95.915,-37.688,179.438,5.406,149.113
C01333=1215.322,-96.165,-37.677,179.436,5.406,149.114
C01334=1215.328,-96.415,-37.667,179.433,5.406,149.114
C01335=1215.333,-96.665,-37.656,179.431,5.406,149.115
C01336=1215.339,-96.915,-37.646,179.429,5.406,149.116
C01337=1215.343,-97.164,-37.635,179.427,5.406,149.116
C01338=1215.349,-97.414,-37.625,179.424,5.405,149.117
C01339=1215.354,-97.664,-37.614,179.422,5.406,149.118
C01340=1215.359,-97.914,-37.604,179.420,5.405,149.118
C01341=1215.364,-98.163,-37.594,179.418,5.406,149.119
C01342=1215.369,-98.413,-37.584,179.415,5.405,149.120
C01343=1215.375,-98.663,-37.574,179.413,5.405,149.120
C01344=1215.380,-98.912,-37.563,179.411,5.405,149.121
C01345=1215.385,-99.162,-37.552,179.409,5.405,149.122
C01346=1215.391,-99.411,-37.542,179.406,5.405,149.122
C01347=1215.396,-99.662,-37.531,179.404,5.405,149.123
C01348=1215.401,-99.911,-37.521,179.402,5.404,149.124
C01349=1215.406,-100.161,-37.511,179.400,5.405,149.124
C01350=1215.411,-100.411,-37.501,179.397,5.404,149.125
C01351=1215.417,-100.682,-37.489,179.394,5.404,149.126
C01352=1215.423,-100.953,-37.479,179.392,5.404,149.127
C01353=1215.429,-101.225,-37.467,179.389,5.404,149.127
C01354=1215.434,-101.496,-37.456,179.387,5.404,149.128
C01355=1215.440,-101.745,-37.446,179.385,5.404,149.129
C01356=1215.445,-101.995,-37.436,179.383,5.404,149.129
C01357=1215.450,-102.245,-37.425,179.380,5.404,149.130
C01358=1215.455,-102.494,-37.416,179.378,5.404,149.131
C01359=1215.460,-102.745,-37.405,179.376,5.403,149.131
C01360=1215.466,-102.994,-37.395,179.373,5.404,149.132
C01361=1215.471,-103.244,-37.385,179.371,5.403,149.133
C01362=1215.476,-103.494,-37.374,179.369,5.404,149.133
C01363=1215.481,-103.743,-37.364,179.366,5.403,149.134
C01364=1215.487,-103.993,-37.354,179.364,5.404,149.135
C01365=1215.492,-104.243,-37.344,179.362,5.403,149.135
C01366=1215.497,-104.493,-37.333,179.360,5.403,149.136
C01367=1215.503,-104.742,-37.323,179.357,5.403,149.137
C01368=1215.507,-104.992,-37.313,179.355,5.403,149.138
C01369=1215.513,-105.242,-37.303,179.352,5.403,149.138
C01370=1215.518,-105.491,-37.293,179.351,5.403,149.139
C01371=1215.523,-105.741,-37.282,179.348,5.402,149.139
C01372=1215.528,-105.991,-37.273,179.346,5.403,149.140
C01373=1215.534,-106.240,-37.262,179.343,5.402,149.141
C01374=1215.539,-106.490,-37.252,179.341,5.403,149.142
C01375=1215.544,-106.740,-37.242,179.339,5.402,149.142
C01376=1215.550,-106.990,-37.233,179.337,5.402,149.143
C01377=1215.555,-107.240,-37.222,179.334,5.402,149.143
C01378=1215.560,-107.490,-37.212,179.332,5.402,149.144
C01379=1215.565,-107.739,-37.202,179.329,5.402,149.145
C01380=1215.571,-107.988,-37.192,179.328,5.402,149.145
C01381=1215.576,-108.239,-37.182,179.325,5.401,149.146
C01382=1215.581,-108.488,-37.171,179.323,5.402,149.147
C01383=1215.586,-108.737,-37.162,179.320,5.401,149.148
C01384=1215.591,-108.988,-37.152,179.318,5.402,149.148
C01385=1215.597,-109.238,-37.142,179.316,5.401,149.149
C01386=1215.602,-109.487,-37.132,179.314,5.401,149.149
C01387=1215.607,-109.737,-37.122,179.311,5.401,149.150
C01388=1215.612,-109.987,-37.111,179.309,5.401,149.151
C01389=1215.618,-110.237,-37.102,179.307,5.401,149.152
C01390=1215.623,-110.486,-37.092,179.305,5.401,149.152
C01391=1215.629,-110.736,-37.082,179.303,5.401,149.153
C01392=1215.633,-110.986,-37.072,179.300,5.401,149.153
C01393=1215.639,-111.235,-37.062,179.298,5.401,149.154
C01394=1215.645,-111.485,-37.052,179.295,5.401,149.155
C01395=1215.649,-111.735,-37.043,179.294,5.401,149.155
C01396=1215.654,-111.985,-37.032,179.291,5.400,149.156
C01397=1215.660,-112.234,-37.022,179.289,5.401,149.157
C01398=1215.665,-112.484,-37.013,179.286,5.400,149.158
C01399=1215.671,-112.734,-37.003,179.284,5.401,149.158
C01400=1215.675,-112.984,-36.993,179.282,5.400,149.159
C01401=1215.681,-113.233,-36.983,179.280,5.400,149.159
C01402=1215.687,-113.483,-36.973,179.277,5.400,149.160
C01403=1215.691,-113.733,-36.964,179.275,5.400,149.161
C01404=1215.697,-113.982,-36.953,179.273,5.399,149.161
C01405=1215.702,-114.233,-36.944,179.271,5.400,149.162
C01406=1215.707,-114.482,-36.934,179.268,5.399,149.163
C01407=1215.713,-114.732,-36.924,179.266,5.400,149.164
C01408=1215.718,-114.982,-36.915,179.263,5.399,149.164
C01409=1215.724,-115.231,-36.905,179.262,5.399,149.165
C01410=1215.728,-115.481,-36.895,179.260,5.400,149.165
C01411=1215.734,-115.731,-36.885,179.257,5.399,149.166
C01412=1215.739,-115.981,-36.875,179.255,5.400,149.167
C01413=1215.744,-116.230,-36.865,179.253,5.399,149.167
C01414=1215.750,-116.480,-36.856,179.251,5.399,149.168
C01415=1215.754,-116.730,-36.846,179.248,5.399,149.169
C01416=1215.760,-116.980,-36.836,179.246,5.399,149.170
C01417=1215.765,-117.230,-36.827,179.243,5.399,149.170
C01418=1215.771,-117.479,-36.816,179.242,5.399,149.171
C01419=1215.776,-117.729,-36.808,179.239,5.398,149.171
C01420=1215.781,-117.979,-36.797,179.237,5.399,149.172
C01421=1215.786,-118.228,-36.787,179.234,5.398,149.173
C01422=1215.792,-118.479,-36.778,179.233,5.398,149.173
C01423=1215.796,-118.728,-36.768,179.230,5.398,149.174
C01424=1215.802,-118.978,-36.759,179.228,5.398,149.175
C01425=1215.807,-119.227,-36.749,179.226,5.399,149.175
C01426=1215.813,-119.477,-36.740,179.224,5.398,149.176
C01427=1215.818,-119.727,-36.730,179.221,5.398,149.177
C01428=1215.823,-119.977,-36.719,179.219,5.398,149.177
C01429=1215.828,-120.227,-36.711,179.217,5.398,149.178
C01430=1215.834,-120.476,-36.700,179.215,5.398,149.179
C01431=1215.839,-120.726,-36.691,179.212,5.398,149.179
C01432=1215.845,-120.976,-36.681,179.210,5.398,149.180
C01433=1215.850,-121.226,-36.672,179.208,5.398,149.181
C01434=1215.855,-121.475,-36.662,179.205,5.397,149.181
C01435=1215.860,-121.725,-36.653,179.203,5.397,149.182
C01436=1215.865,-121.975,-36.643,179.201,5.397,149.183
C01437=1215.871,-122.225,-36.634,179.199,5.397,149.183
C01438=1215.875,-122.474,-36.624,179.197,5.397,149.184
C01439=1215.881,-122.724,-36.615,179.194,5.397,149.185
C01440=1215.886,-122.974,-36.605,179.192,5.397,149.185
C01441=1215.892,-123.224,-36.596,179.190,5.397,149.186
C01442=1215.897,-123.473,-36.586,179.188,5.397,149.187
C01443=1215.902,-123.723,-36.577,179.185,5.397,149.187
C01444=1215.908,-123.973,-36.568,179.183,5.397,149.188
C01445=1215.913,-124.222,-36.558,179.180,5.397,149.189
C01446=1215.919,-124.472,-36.548,179.179,5.397,149.189
C01447=1215.923,-124.722,-36.538,179.176,5.396,149.190
C01448=1215.928,-124.972,-36.530,179.174,5.397,149.191
C01449=1215.934,-125.222,-36.519,179.172,5.397,149.191
C01450=1215.939,-125.472,-36.510,179.170,5.396,149.192
C01451=1215.944,-125.721,-36.502,179.168,5.397,149.193
C01452=1215.950,-125.971,-36.491,179.165,5.396,149.193
C01453=1215.955,-126.221,-36.482,179.163,5.396,149.194
C01454=1215.961,-126.471,-36.473,179.161,5.396,149.194
C01455=1215.538,-126.481,-36.510,179.156,5.399,149.197
C01456=1215.533,-126.232,-36.519,179.159,5.400,149.196
C01457=1215.528,-125.982,-36.528,179.161,5.399,149.195
C01458=1215.523,-125.732,-36.538,179.164,5.400,149.194
C01459=1215.518,-125.482,-36.548,179.165,5.400,149.194
C01460=1215.513,-125.232,-36.557,179.168,5.400,149.193
C01461=1215.507,-124.982,-36.566,179.170,5.400,149.192
C01462=1215.502,-124.733,-36.576,179.172,5.400,149.192
C01463=1215.496,-124.483,-36.585,179.174,5.400,149.191
C01464=1215.492,-124.234,-36.595,179.177,5.400,149.191
C01465=1215.486,-123.984,-36.604,179.179,5.400,149.190
C01466=1215.480,-123.734,-36.613,179.181,5.400,149.189
C01467=1215.476,-123.484,-36.623,179.184,5.401,149.189
C01468=1215.470,-123.234,-36.633,179.186,5.400,149.188
C01469=1215.465,-122.985,-36.642,179.188,5.401,149.187
C01470=1215.460,-122.735,-36.651,179.190,5.401,149.187
C01471=1215.455,-122.485,-36.662,179.193,5.401,149.186
C01472=1215.449,-122.235,-36.670,179.195,5.401,149.185
C01473=1215.444,-121.986,-36.681,179.197,5.400,149.185
C01474=1215.439,-121.736,-36.690,179.199,5.401,149.184
C01475=1215.433,-121.486,-36.700,179.201,5.401,149.183
C01476=1215.428,-121.236,-36.709,179.204,5.401,149.183
C01477=1215.422,-120.987,-36.719,179.206,5.401,149.182
C01478=1215.417,-120.737,-36.728,179.208,5.401,149.181
C01479=1215.412,-120.488,-36.737,179.210,5.401,149.181
C01480=1215.407,-120.237,-36.747,179.213,5.401,149.180
C01481=1215.402,-119.988,-36.757,179.215,5.401,149.179
C01482=1215.396,-119.737,-36.766,179.217,5.402,149.179
C01483=1215.391,-119.488,-36.776,179.219,5.402,149.178
C01484=1215.385,-119.238,-36.786,179.222,5.402,149.177
C01485=1215.381,-118.989,-36.795,179.224,5.402,149.177
C01486=1215.375,-118.739,-36.805,179.225,5.402,149.176
C01487=1215.370,-118.489,-36.815,179.228,5.402,149.175
C01488=1215.365,-118.239,-36.825,179.230,5.402,149.175
C01489=1215.360,-117.989,-36.834,179.233,5.402,149.174
C01490=1215.354,-117.740,-36.844,179.235,5.402,149.174
C01491=1215.349,-117.490,-36.853,179.237,5.402,149.173
C01492=1215.343,-117.240,-36.863,179.239,5.402,149.172
C01493=1215.339,-116.990,-36.873,179.242,5.402,149.171
C01494=1215.333,-116.740,-36.882,179.244,5.402,149.171
C01495=1215.328,-116.491,-36.892,179.246,5.403,149.170
C01496=1215.323,-116.241,-36.902,179.248,5.402,149.169
C01497=1215.317,-115.991,-36.912,179.251,5.403,149.169
C01498=1215.312,-115.742,-36.921,179.253,5.402,149.168
C01499=1215.307,-115.492,-36.932,179.255,5.403,149.168
C01500=1215.302,-115.242,-36.941,179.257,5.403,149.167
C01501=1215.296,-114.992,-36.951,179.260,5.403,149.166
C01502=1215.291,-114.743,-36.961,179.262,5.403,149.165
C01503=1215.285,-114.493,-36.970,179.264,5.403,149.165
C01504=1215.280,-114.243,-36.981,179.266,5.403,149.164
C01505=1215.276,-113.994,-36.990,179.269,5.403,149.163
C01506=1215.270,-113.743,-37.000,179.271,5.403,149.163
C01507=1215.265,-113.494,-37.009,179.273,5.403,149.162
C01508=1215.259,-113.245,-37.020,179.276,5.404,149.162
C01509=1215.254,-112.994,-37.030,179.278,5.403,149.161
C01510=1215.249,-112.745,-37.039,179.280,5.404,149.160
C01511=1215.243,-112.495,-37.049,179.282,5.403,149.159
C01512=1215.239,-112.246,-37.059,179.285,5.404,149.159
C01513=1215.233,-111.995,-37.069,179.287,5.404,149.158
C01514=1215.228,-111.745,-37.079,179.289,5.404,149.158
C01515=1215.223,-111.496,-37.089,179.291,5.404,149.157
C01516=1215.217,-111.247,-37.099,179.294,5.404,149.156
C01517=1215.211,-110.996,-37.108,179.296,5.404,149.156
C01518=1215.207,-110.746,-37.118,179.298,5.405,149.155
C01519=1215.201,-110.497,-37.129,179.300,5.404,149.154
C01520=1215.196,-110.247,-37.139,179.303,5.404,149.153
C01521=1215.191,-109.998,-37.148,179.305,5.405,149.153
C01522=1215.186,-109.747,-37.158,179.307,5.404,149.152
C01523=1215.180,-109.498,-37.168,179.310,5.405,149.152
C01524=1215.175,-109.249,-37.178,179.312,5.404,149.151
C01525=1215.170,-108.998,-37.189,179.314,5.405,149.150
C01526=1215.165,-108.749,-37.199,179.316,5.405,149.150
C01527=1215.159,-108.499,-37.208,179.319,5.405,149.149
C01528=1215.154,-108.249,-37.218,179.321,5.405,149.148
C01529=1215.149,-107.999,-37.229,179.323,5.405,149.147
C01530=1215.144,-107.750,-37.238,179.325,5.405,149.147
C01531=1215.138,-107.500,-37.248,179.328,5.406,149.146
C01532=1215.133,-107.250,-37.259,179.330,5.405,149.146
C01533=1215.128,-107.001,-37.269,179.332,5.406,149.145
C01534=1215.123,-106.751,-37.278,179.334,5.405,149.144
C01535=1215.117,-106.501,-37.288,179.337,5.406,149.143
C01536=1215.112,-106.251,-37.299,179.339,5.406,149.143
C01537=1215.107,-106.002,-37.308,179.341,5.406,149.142
C01538=1215.102,-105.752,-37.319,179.344,5.406,149.142
C01539=1215.097,-105.502,-37.329,179.346,5.406,149.141
C01540=1215.091,-105.252,-37.339,179.348,5.406,149.140
C01541=1215.086,-105.003,-37.349,179.350,5.407,149.140
C01542=1215.081,-104.753,-37.360,179.353,5.406,149.139
C01543=1215.076,-104.503,-37.370,179.355,5.407,149.138
C01544=1215.070,-104.254,-37.380,179.357,5.406,149.137
C01545=1215.065,-104.004,-37.391,179.360,5.407,149.137
C01546=1215.060,-103.754,-37.400,179.362,5.406,149.136
C01547=1215.054,-103.505,-37.410,179.364,5.407,149.136
C01548=1215.049,-103.255,-37.421,179.366,5.407,149.135
C01549=1215.044,-103.005,-37.431,179.369,5.407,149.134
C01550=1215.039,-102.756,-37.441,179.371,5.407,149.133
C01551=1215.034,-102.505,-37.451,179.374,5.407,149.133
C01552=1215.028,-102.256,-37.462,179.375,5.407,149.132
C01553=1215.023,-102.006,-37.472,179.378,5.408,149.131
C01554=1215.018,-101.756,-37.482,179.380,5.407,149.131
C01555=1215.012,-101.507,-37.493,179.383,5.408,149.130
C01556=1215.007,-101.235,-37.504,179.385,5.407,149.129
C01557=1215.002,-100.964,-37.514,179.388,5.408,149.129
C01558=1214.995,-100.693,-37.526,179.390,5.407,149.128
C01559=1214.990,-100.422,-37.537,179.392,5.408,149.127
C01560=1214.985,-100.172,-37.547,179.395,5.408,149.126
C01561=1214.980,-99.922,-37.557,179.397,5.408,149.126
C01562=1214.974,-99.672,-37.568,179.400,5.408,149.125
C01563=1214.969,-99.422,-37.578,179.401,5.408,149.125
C01564=1214.963,-99.173,-37.588,179.404,5.409,149.124
C01565=1214.958,-98.922,-37.599,179.406,5.408,149.123
C01566=1214.954,-98.673,-37.609,179.409,5.409,149.122
C01567=1214.948,-98.424,-37.619,179.411,5.408,149.122
C01568=1214.943,-98.174,-37.630,179.414,5.409,149.121
C01569=1214.938,-97.925,-37.640,179.415,5.409,149.121
C01570=1214.933,-97.674,-37.651,179.418,5.409,149.120
C01571=1214.927,-97.425,-37.661,179.420,5.409,149.119
C01572=1214.921,-97.175,-37.671,179.423,5.409,149.118
C01573=1214.916,-96.925,-37.682,179.425,5.409,149.118
C01574=1214.911,-96.676,-37.693,179.427,5.409,149.117
C01575=1214.906,-96.426,-37.703,179.429,5.409,149.117
C01576=1214.901,-96.176,-37.714,179.432,5.410,149.116
C01577=1214.896,-95.926,-37.724,179.434,5.410,149.115
C01578=1214.890,-95.676,-37.734,179.436,5.410,149.114
C01579=1214.885,-95.427,-37.744,179.439,5.410,149.114
C01580=1214.880,-95.178,-37.755,179.441,5.410,149.113
C01581=1214.875,-94.928,-37.765,179.443,5.410,149.112
C01582=1214.870,-94.678,-37.776,179.446,5.410,149.112
C01583=1214.864,-94.428,-37.786,179.448,5.410,149.111
C01584=1214.859,-94.178,-37.797,179.450,5.411,149.110
C01585=1214.854,-93.929,-37.808,179.452,5.410,149.110
C01586=1214.849,-93.679,-37.818,179.455,5.411,149.109
C01587=1214.843,-93.429,-37.829,179.457,5.410,149.108
C01588=1214.838,-93.179,-37.839,179.459,5.411,149.108
C01589=1214.833,-92.930,-37.850,179.461,5.411,149.107
C01590=1214.828,-92.680,-37.861,179.464,5.411,149.106
C01591=1214.822,-92.430,-37.871,179.466,5.411,149.106
C01592=1214.817,-92.180,-37.881,179.469,5.411,149.105
C01593=1214.812,-91.931,-37.892,179.471,5.411,149.104
C01594=1214.807,-91.681,-37.903,179.473,5.412,149.104
C01595=1214.802,-91.431,-37.913,179.475,5.411,149.103
C01596=1214.797,-91.182,-37.924,179.478,5.412,149.102
C01597=1214.791,-90.932,-37.935,179.480,5.411,149.102
C01598=1214.786,-90.682,-37.945,179.483,5.412,149.101
C01599=1214.781,-90.433,-37.956,179.485,5.411,149.100
C01600=1214.775,-90.182,-37.967,179.487,5.412,149.099
C01601=1214.770,-89.933,-37.977,179.489,5.412,149.099
C01602=1214.765,-89.683,-37.989,179.492,5.412,149.098
C01603=1214.759,-89.434,-37.999,179.494,5.412,149.097
C01604=1214.754,-89.184,-38.010,179.496,5.412,149.097
C01605=1214.749,-88.935,-38.020,179.499,5.413,149.096
C01606=1214.744,-88.684,-38.031,179.501,5.412,149.095
C01607=1214.738,-88.435,-38.041,179.504,5.413,149.095
C01608=1214.734,-88.185,-38.053,179.505,5.413,149.094
C01609=1214.728,-87.936,-38.063,179.508,5.413,149.093
C01610=1214.723,-87.686,-38.074,179.510,5.413,149.093
C01611=1214.718,-87.436,-38.085,179.513,5.413,149.092
C01612=1214.713,-87.186,-38.095,179.515,5.413,149.091
C01613=1214.707,-86.936,-38.107,179.518,5.413,149.091
C01614=1214.702,-86.687,-38.117,179.520,5.413,149.090
C01615=1214.697,-86.437,-38.128,179.522,5.414,149.089
C01616=1214.692,-86.188,-38.138,179.524,5.413,149.089
C01617=1214.687,-85.938,-38.150,179.527,5.414,149.088
C01618=1214.682,-85.688,-38.160,179.529,5.414,149.087
C01619=1214.677,-85.439,-38.171,179.531,5.414,149.087
C01620=1214.672,-85.189,-38.182,179.534,5.414,149.086
C01621=1214.666,-84.939,-38.193,179.536,5.414,149.085
C01622=1214.661,-84.689,-38.204,179.538,5.414,149.084
C01623=1214.656,-84.439,-38.215,179.540,5.415,149.084
C01624=1214.650,-84.190,-38.225,179.543,5.415,149.083
C01625=1214.646,-83.940,-38.237,179.545,5.415,149.083
C01626=1214.640,-83.691,-38.247,179.548,5.415,149.082
C01627=1214.635,-83.441,-38.259,179.550,5.415,149.081
C01628=1214.630,-83.191,-38.269,179.553,5.415,149.080
C01629=1214.624,-82.942,-38.280,179.555,5.415,149.080
C01630=1214.619,-82.691,-38.291,179.557,5.416,149.079
C01631=1214.615,-82.442,-38.302,179.559,5.415,149.079
C01632=1214.608,-82.192,-38.313,179.562,5.416,149.078
C01633=1214.604,-81.942,-38.324,179.564,5.415,149.077
C01634=1214.598,-81.693,-38.334,179.566,5.416,149.076
C01635=1214.593,-81.443,-38.346,179.569,5.415,149.076
C01636=1214.589,-81.193,-38.357,179.571,5.416,149.075
C01637=1214.582,-80.944,-38.368,179.574,5.416,149.074
C01638=1214.578,-80.694,-38.379,179.576,5.416,149.074
C01639=1214.573,-80.444,-38.390,179.578,5.417,149.073
C01640=1214.567,-80.195,-38.401,179.580,5.416,149.072
C01641=1214.562,-79.945,-38.412,179.583,5.417,149.072
C01642=1214.557,-79.695,-38.423,179.585,5.416,149.071
C01643=1214.552,-79.446,-38.434,179.588,5.417,149.070
C01644=1214.547,-79.195,-38.445,179.590,5.416,149.070
C01645=1214.541,-78.946,-38.456,179.592,5.417,149.069
C01646=1214.536,-78.697,-38.467,179.595,5.417,149.068
C01647=1214.531,-78.446,-38.478,179.597,5.417,149.068
C01648=1214.525,-78.196,-38.490,179.599,5.418,149.067
C01649=1214.520,-77.948,-38.501,179.601,5.417,149.066
C01650=1214.515,-77.697,-38.511,179.604,5.418,149.066
C01651=1214.510,-77.447,-38.523,179.606,5.418,149.065
C01652=1214.504,-77.198,-38.534,179.609,5.418,149.064
C01653=1214.499,-76.948,-38.545,179.611,5.418,149.063
C01654=1214.495,-76.699,-38.556,179.614,5.418,149.063
C01655=1214.489,-76.449,-38.567,179.615,5.418,149.062
C01656=1214.484,-76.200,-38.579,179.618,5.419,149.061
C01657=1214.478,-75.949,-38.590,179.621,5.419,149.061
C01658=1214.474,-75.699,-38.601,179.623,5.419,149.060
C01659=1214.468,-75.451,-38.612,179.625,5.419,149.059
C01660=1214.463,-75.180,-38.624,179.627,5.419,149.059
C01661=1214.457,-74.909,-38.637,179.630,5.419,149.058
C01662=1214.451,-74.638,-38.649,179.633,5.420,149.057
C01663=1214.445,-74.368,-38.662,179.635,5.419,149.056
C01664=1214.440,-74.118,-38.672,179.638,5.420,149.056
C01665=1214.435,-73.869,-38.683,179.640,5.419,149.055
C01666=1214.430,-73.619,-38.695,179.642,5.420,149.054
C01667=1214.425,-73.369,-38.706,179.645,5.420,149.054
C01668=1214.420,-73.120,-38.717,179.647,5.420,149.053
C01669=1214.414,-72.870,-38.728,179.650,5.420,149.052
C01670=1214.409,-72.620,-38.740,179.652,5.420,149.052
C01671=1214.404,-72.370,-38.751,179.655,5.420,149.051
C01672=1214.399,-72.121,-38.762,179.657,5.420,149.050
C01673=1214.393,-71.871,-38.774,179.659,5.421,149.050
C01674=1214.388,-71.622,-38.786,179.661,5.421,149.049
C01675=1214.383,-71.371,-38.796,179.664,5.421,149.048
C01676=1214.378,-71.122,-38.808,179.666,5.421,149.048
C01677=1214.373,-70.873,-38.819,179.668,5.421,149.047
C01678=1214.367,-70.623,-38.831,179.671,5.422,149.046
C01679=1214.363,-70.373,-38.842,179.673,5.421,149.045
C01680=1214.357,-70.123,-38.854,179.676,5.422,149.045
C01681=1214.352,-69.874,-38.865,179.678,5.422,149.044
C01682=1214.347,-69.624,-38.877,179.680,5.422,149.043
C01683=1214.342,-69.375,-38.888,179.683,5.423,149.043
C01684=1214.336,-69.124,-38.899,179.685,5.422,149.042
C01685=1214.331,-68.874,-38.911,179.687,5.423,149.041
C01686=1214.326,-68.626,-38.921,179.689,5.422,149.041
C01687=1214.321,-68.376,-38.933,179.692,5.423,149.040
C01688=1214.316,-68.126,-38.945,179.695,5.423,149.039
C01689=1214.311,-67.876,-38.957,179.697,5.423,149.039
C01690=1214.306,-67.626,-38.968,179.700,5.423,149.038
C01691=1214.300,-67.376,-38.980,179.702,5.423,149.037
C01692=1214.294,-67.127,-38.991,179.704,5.423,149.036
C01693=1214.290,-66.878,-39.003,179.706,5.423,149.036
C01694=1214.284,-66.628,-39.014,179.709,5.424,149.035
C01695=1214.280,-66.378,-39.026,179.711,5.424,149.035
C01696=1214.274,-66.128,-39.038,179.713,5.424,149.034
C01697=1214.269,-65.878,-39.049,179.716,5.424,149.033
C01698=1214.263,-65.629,-39.060,179.718,5.424,149.032
C01699=1214.259,-65.380,-39.072,179.721,5.425,149.032
C01700=1214.253,-65.130,-39.084,179.723,5.424,149.031
C01701=1214.249,-64.880,-39.095,179.726,5.425,149.030
C01702=1214.243,-64.630,-39.107,179.728,5.425,149.030
C01703=1214.238,-64.380,-39.119,179.730,5.425,149.029
C01704=1214.233,-64.131,-39.130,179.732,5.426,149.028
C01705=1214.227,-63.881,-39.141,179.735,5.425,149.028
C01706=1214.222,-63.632,-39.153,179.737,5.426,149.027
C01707=1214.217,-63.382,-39.165,179.740,5.426,149.026
C01708=1214.213,-63.133,-39.177,179.742,5.426,149.026
C01709=1214.207,-62.883,-39.189,179.745,5.426,149.025
C01710=1214.202,-62.633,-39.200,179.747,5.426,149.024
C01711=1214.197,-62.383,-39.212,179.749,5.426,149.023
C01712=1214.192,-62.133,-39.224,179.752,5.427,149.023
C01713=1214.187,-61.884,-39.235,179.754,5.426,149.022
C01714=1214.181,-61.634,-39.246,179.756,5.427,149.022
C01715=1214.175,-61.385,-39.258,179.758,5.427,149.021
C01716=1214.171,-61.136,-39.270,179.761,5.427,149.020
C01717=1214.166,-60.886,-39.282,179.764,5.428,149.019
C01718=1214.160,-60.636,-39.294,179.766,5.427,149.019
C01719=1214.155,-60.386,-39.305,179.769,5.428,149.018
C01720=1214.150,-60.136,-39.317,179.771,5.428,149.017
C01721=1214.145,-59.886,-39.329,179.773,5.428,149.017
C01722=1214.140,-59.637,-39.341,179.775,5.428,149.016
C01723=1214.135,-59.387,-39.353,179.778,5.428,149.015
C01724=1214.129,-59.137,-39.365,179.781,5.429,149.015
C01725=1214.125,-58.888,-39.376,179.783,5.428,149.014
C01726=1214.119,-58.638,-39.388,179.785,5.429,149.013
C01727=1214.114,-58.388,-39.401,179.788,5.430,149.013
C01728=1214.109,-58.139,-39.412,179.790,5.429,149.012
C01729=1214.103,-57.890,-39.423,179.792,5.430,149.011
C01730=1214.098,-57.640,-39.435,179.794,5.429,149.011
C01731=1214.094,-57.391,-39.447,179.797,5.430,149.010
C01732=1214.088,-57.141,-39.459,179.800,5.430,149.009
C01733=1214.083,-56.891,-39.471,179.802,5.430,149.008
C01734=1214.078,-56.641,-39.484,179.805,5.430,149.008
C01735=1214.073,-56.392,-39.495,179.807,5.430,149.007
C01736=1214.067,-56.142,-39.507,179.809,5.430,149.006
C01737=1214.062,-55.892,-39.519,179.812,5.431,149.006
C01738=1214.057,-55.643,-39.531,179.814,5.431,149.005
C01739=1214.052,-55.393,-39.543,179.816,5.431,149.004
C01740=1214.047,-55.143,-39.555,179.818,5.431,149.004
C01741=1214.042,-54.894,-39.567,179.821,5.432,149.003
C01742=1214.036,-54.644,-39.579,179.824,5.432,149.002
C01743=1214.032,-54.394,-39.590,179.826,5.432,149.002
C01744=1214.026,-54.145,-39.603,179.828,5.432,149.001
C01745=1214.021,-53.895,-39.615,179.830,5.432,149.000
C01746=1214.016,-53.645,-39.627,179.833,5.432,149.000
C01747=1214.011,-53.396,-39.639,179.836,5.433,148.999
C01748=1214.006,-53.146,-39.651,179.838,5.432,148.998
C01749=1214.001,-52.897,-39.663,179.841,5.433,148.997
C01750=1213.996,-52.646,-39.675,179.843,5.433,148.997
C01751=1213.990,-52.396,-39.687,179.845,5.433,148.996
C01752=1213.986,-52.147,-39.699,179.847,5.434,148.996
C01753=1213.981,-51.897,-39.711,179.850,5.433,148.995
C01754=1213.975,-51.648,-39.724,179.852,5.434,148.994
C01755=1213.970,-51.398,-39.736,179.855,5.434,148.993
C01756=1213.965,-51.148,-39.748,179.857,5.434,148.993
C01757=1213.959,-50.899,-39.760,179.860,5.435,148.992
C01758=1213.955,-50.649,-39.771,179.862,5.435,148.991
C01759=1213.950,-50.400,-39.784,179.864,5.435,148.991
C01760=1213.944,-50.150,-39.796,179.867,5.435,148.990
C01761=1213.939,-49.900,-39.809,179.869,5.435,148.989
C01762=1213.934,-49.651,-39.820,179.872,5.435,148.989
C01763=1213.929,-49.401,-39.833,179.874,5.436,148.988
C01764=1213.923,-49.131,-39.846,179.877,5.435,148.987
C01765=1213.917,-48.861,-39.859,179.879,5.436,148.986
C01766=1213.912,-48.591,-39.872,179.882,5.436,148.986
C01767=1213.906,-48.321,-39.886,179.885,5.437,148.985
C01768=1213.901,-48.071,-39.898,179.887,5.436,148.984
C01769=1213.896,-47.822,-39.910,179.889,5.437,148.984
C01770=1213.891,-47.573,-39.922,179.892,5.437,148.983
C01771=1213.886,-47.323,-39.934,179.894,5.437,148.982
C01772=1213.881,-47.073,-39.947,179.897,5.437,148.981
C01773=1213.875,-46.823,-39.959,179.899,5.438,148.981
C01774=1213.870,-46.574,-39.971,179.901,5.438,148.980
C01775=1213.865,-46.323,-39.984,179.904,5.438,148.979
C01776=1213.860,-46.074,-39.996,179.906,5.438,148.979
C01777=1213.855,-45.825,-40.009,179.908,5.439,148.978
C01778=1213.850,-45.575,-40.021,179.911,5.439,148.977
C01779=1213.845,-45.326,-40.033,179.913,5.439,148.977
C01780=1213.839,-45.076,-40.045,179.916,5.439,148.976
C01781=1213.834,-44.826,-40.058,179.918,5.440,148.975
C01782=1213.829,-44.577,-40.070,179.921,5.439,148.975
C01783=1213.824,-44.326,-40.083,179.923,5.440,148.974
C01784=1213.819,-44.077,-40.095,179.926,5.440,148.973
C01785=1213.814,-43.828,-40.108,179.928,5.440,148.973
C01786=1213.808,-43.578,-40.120,179.931,5.440,148.972
C01787=1213.803,-43.328,-40.132,179.933,5.441,148.971
C01788=1213.798,-43.079,-40.145,179.935,5.441,148.970
C01789=1213.793,-42.828,-40.157,179.938,5.441,148.970
C01790=1213.788,-42.579,-40.170,179.940,5.442,148.969
C01791=1213.783,-42.330,-40.182,179.942,5.442,148.969
C01792=1213.778,-42.080,-40.194,179.945,5.442,148.968
C01793=1213.773,-41.831,-40.207,179.947,5.442,148.967
C01794=1213.767,-41.581,-40.219,179.950,5.442,148.966
C01795=1213.763,-41.331,-40.232,179.952,5.443,148.966
C01796=1213.757,-41.081,-40.244,179.954,5.442,148.965
C01797=1213.752,-40.832,-40.257,179.957,5.443,148.964
C01798=1213.747,-40.583,-40.269,179.960,5.443,148.964
C01799=1213.742,-40.333,-40.282,179.962,5.443,148.963
C01800=1213.737,-40.083,-40.294,179.965,5.443,148.962
C01801=1213.732,-39.833,-40.307,179.967,5.444,148.962
C01802=1213.727,-39.584,-40.320,179.969,5.443,148.961
C01803=1213.721,-39.334,-40.333,179.972,5.444,148.960
C01804=1213.716,-39.084,-40.345,179.974,5.445,148.960
C01805=1213.711,-38.834,-40.358,179.976,5.444,148.959
C01806=1213.706,-38.585,-40.370,179.979,5.445,148.958
C01807=1213.701,-38.336,-40.383,179.982,5.445,148.958
C01808=1213.696,-38.087,-40.395,179.984,5.445,148.957
C01809=1213.691,-37.836,-40.408,179.986,5.446,148.956
C01810=1213.686,-37.587,-40.420,179.989,5.446,148.956
C01811=1213.680,-37.337,-40.433,179.991,5.446,148.955
C01812=1213.675,-37.088,-40.446,179.994,5.446,148.954
C01813=1213.670,-36.838,-40.459,179.996,5.447,148.953
C01814=1213.665,-36.588,-40.472,179.998,5.446,148.953
C01815=1213.660,-36.339,-40.484,-179.999,5.447,148.952
C01816=1213.655,-36.089,-40.496,-179.996,5.447,148.951
C01817=1213.650,-35.839,-40.509,-179.994,5.447,148.951
C01818=1213.644,-35.589,-40.522,-179.992,5.448,148.950
C01819=1213.639,-35.340,-40.535,-179.989,5.448,148.949
C01820=1213.634,-35.091,-40.547,-179.987,5.448,148.949
C01821=1213.630,-34.841,-40.560,-179.985,5.448,148.948
C01822=1213.624,-34.591,-40.573,-179.982,5.449,148.947
C01823=1213.619,-34.342,-40.586,-179.980,5.449,148.947
C01824=1213.613,-34.092,-40.599,-179.977,5.449,148.946
C01825=1213.609,-33.842,-40.612,-179.975,5.450,148.945
C01826=1213.604,-33.593,-40.624,-179.972,5.449,148.945
C01827=1213.599,-33.344,-40.637,-179.970,5.450,148.944
